	CELL_LC401_AP_TH_D02                            :=      47382       ,
	CELL_LC401_AP_TH_D03                            :=      47383       ,
	CELL_LC401_AP_TH_D04                            :=      47384       ,
	CELL_LC501_TESTER                               :=      47400       ,
	CELL_LC501_TESTER_SOCKET_A01                    :=      47401       ,
	CELL_LC501_TESTER_SOCKET_A02                    :=      47402       ,
	CELL_LC501_TESTER_SOCKET_A03                    :=      47403       ,
	CELL_LC501_TESTER_SOCKET_A04                    :=      47404       ,
	CELL_LC501_TESTER_SOCKET_B01                    :=      47411       ,
	CELL_LC501_TESTER_SOCKET_B02                    :=      47412       ,
	CELL_LC501_TESTER_SOCKET_B03                    :=      47413       ,
	CELL_LC501_TESTER_SOCKET_B04                    :=      47414       ,
	CELL_LC501_TESTER_SOCKET_C01                    :=      47421       ,
	CELL_LC501_TESTER_SOCKET_C02                    :=      47422       ,
	CELL_LC501_TESTER_SOCKET_C03                    :=      47423       ,
	CELL_LC501_TESTER_SOCKET_C04                    :=      47424       ,
	CELL_LC501_TESTER_SOCKET_D01                    :=      47431       ,
	CELL_LC501_TESTER_SOCKET_D02                    :=      47432       ,
	CELL_LC501_TESTER_SOCKET_D03                    :=      47433       ,
	CELL_LC501_TESTER_SOCKET_D04                    :=      47434       ,
	CELL_LC501_AP                                   :=      47450       ,
	CELL_LC501_AP_TH_A01                            :=      47451       ,
	CELL_LC501_AP_TH_A02                            :=      47452       ,
	CELL_LC501_AP_TH_A03                            :=      47453       ,
	CELL_LC501_AP_TH_A04                            :=      47454       ,
	CELL_LC501_AP_TH_B01                            :=      47461       ,
	CELL_LC501_AP_TH_B02                            :=      47462       ,
	CELL_LC501_AP_TH_B03                            :=      47463       ,
	CELL_LC501_AP_TH_B04                            :=      47464       ,
	CELL_LC501_AP_TH_C01                            :=      47471       ,
	CELL_LC501_AP_TH_C02                            :=      47472       ,
	CELL_LC501_AP_TH_C03                            :=      47473       ,
	CELL_LC501_AP_TH_C04                            :=      47474       ,
	CELL_LC501_AP_TH_D01                            :=      47481       ,
	CELL_LC501_AP_TH_D02                            :=      47482       ,
	CELL_LC501_AP_TH_D03                            :=      47483       ,
	CELL_LC501_AP_TH_D04                            :=      47484       ,
	CELL_LC601_TESTER                               :=      47500       ,
	CELL_LC601_TESTER_SOCKET_A01                    :=      47501       ,
	CELL_LC601_TESTER_SOCKET_A02                    :=      47502       ,
	CELL_LC601_TESTER_SOCKET_A03                    :=      47503       ,
	CELL_LC601_TESTER_SOCKET_A04                    :=      47504       ,
	CELL_LC601_TESTER_SOCKET_B01                    :=      47511       ,
	CELL_LC601_TESTER_SOCKET_B02                    :=      47512       ,
	CELL_LC601_TESTER_SOCKET_B03                    :=      47513       ,
	CELL_LC601_TESTER_SOCKET_B04                    :=      47514       ,
	CELL_LC601_TESTER_SOCKET_C01                    :=      47521       ,
	CELL_LC601_TESTER_SOCKET_C02                    :=      47522       ,
	CELL_LC601_TESTER_SOCKET_C03                    :=      47523       ,
	CELL_LC601_TESTER_SOCKET_C04                    :=      47524       ,
	CELL_LC601_TESTER_SOCKET_D01                    :=      47531       ,
	CELL_LC601_TESTER_SOCKET_D02                    :=      47532       ,
	CELL_LC601_TESTER_SOCKET_D03                    :=      47533       ,
	CELL_LC601_TESTER_SOCKET_D04                    :=      47534       ,
	CELL_LC601_AP                                   :=      47550       ,
	CELL_LC601_AP_TH_A01                            :=      47551       ,
	CELL_LC601_AP_TH_A02                            :=      47552       ,
	CELL_LC601_AP_TH_A03                            :=      47553       ,
	CELL_LC601_AP_TH_A04                            :=      47554       ,
	CELL_LC601_AP_TH_B01                            :=      47561       ,
	CELL_LC601_AP_TH_B02                            :=      47562       ,
	CELL_LC601_AP_TH_B03                            :=      47563       ,
	CELL_LC601_AP_TH_B04                            :=      47564       ,
	CELL_LC601_AP_TH_C01                            :=      47571       ,
	CELL_LC601_AP_TH_C02                            :=      47572       ,
	CELL_LC601_AP_TH_C03                            :=      47573       ,
	CELL_LC601_AP_TH_C04                            :=      47574       ,
	CELL_LC601_AP_TH_D01                            :=      47581       ,
	CELL_LC601_AP_TH_D02                            :=      47582       ,
	CELL_LC601_AP_TH_D03                            :=      47583       ,
	CELL_LC601_AP_TH_D04                            :=      47584       ,
	CELL_RA101_TESTER                               :=      50000       ,
	CELL_RA101_TESTER_SOCKET_A01                    :=      50001       ,
	CELL_RA101_TESTER_SOCKET_A02                    :=      50002       ,
	CELL_RA101_TESTER_SOCKET_A03                    :=      50003       ,
	CELL_RA101_TESTER_SOCKET_A04                    :=      50004       ,
	CELL_RA101_TESTER_SOCKET_B01                    :=      50011       ,
	CELL_RA101_TESTER_SOCKET_B02                    :=      50012       ,
	CELL_RA101_TESTER_SOCKET_B03                    :=      50013       ,
	CELL_RA101_TESTER_SOCKET_B04                    :=      50014       ,
	CELL_RA101_TESTER_SOCKET_C01                    :=      50021       ,
	CELL_RA101_TESTER_SOCKET_C02                    :=      50022       ,
	CELL_RA101_TESTER_SOCKET_C03                    :=      50023       ,
	CELL_RA101_TESTER_SOCKET_C04                    :=      50024       ,
	CELL_RA101_TESTER_SOCKET_D01                    :=      50031       ,
	CELL_RA101_TESTER_SOCKET_D02                    :=      50032       ,
	CELL_RA101_TESTER_SOCKET_D03                    :=      50033       ,
	CELL_RA101_TESTER_SOCKET_D04                    :=      50034       ,
	CELL_RA101_AP                                   :=      50050       ,
	CELL_RA101_AP_TH_A01                            :=      50051       ,
	CELL_RA101_AP_TH_A02                            :=      50052       ,
	CELL_RA101_AP_TH_A03                            :=      50053       ,
	CELL_RA101_AP_TH_A04                            :=      50054       ,
	CELL_RA101_AP_TH_B01                            :=      50061       ,
	CELL_RA101_AP_TH_B02                            :=      50062       ,
	CELL_RA101_AP_TH_B03                            :=      50063       ,
	CELL_RA101_AP_TH_B04                            :=      50064       ,
	CELL_RA101_AP_TH_C01                            :=      50071       ,
	CELL_RA101_AP_TH_C02                            :=      50072       ,
	CELL_RA101_AP_TH_C03                            :=      50073       ,
	CELL_RA101_AP_TH_C04                            :=      50074       ,
	CELL_RA101_AP_TH_D01                            :=      50081       ,
	CELL_RA101_AP_TH_D02                            :=      50082       ,
	CELL_RA101_AP_TH_D03                            :=      50083       ,
	CELL_RA101_AP_TH_D04                            :=      50084       ,
	CELL_RA201_TESTER                               :=      50100       ,
	CELL_RA201_TESTER_SOCKET_A01                    :=      50101       ,
	CELL_RA201_TESTER_SOCKET_A02                    :=      50102       ,
	CELL_RA201_TESTER_SOCKET_A03                    :=      50103       ,
	CELL_RA201_TESTER_SOCKET_A04                    :=      50104       ,
	CELL_RA201_TESTER_SOCKET_B01                    :=      50111       ,
	CELL_RA201_TESTER_SOCKET_B02                    :=      50112       ,
	CELL_RA201_TESTER_SOCKET_B03                    :=      50113       ,
	CELL_RA201_TESTER_SOCKET_B04                    :=      50114       ,
	CELL_RA201_TESTER_SOCKET_C01                    :=      50121       ,
	CELL_RA201_TESTER_SOCKET_C02                    :=      50122       ,
	CELL_RA201_TESTER_SOCKET_C03                    :=      50123       ,
	CELL_RA201_TESTER_SOCKET_C04                    :=      50124       ,
	CELL_RA201_TESTER_SOCKET_D01                    :=      50131       ,
	CELL_RA201_TESTER_SOCKET_D02                    :=      50132       ,
	CELL_RA201_TESTER_SOCKET_D03                    :=      50133       ,
	CELL_RA201_TESTER_SOCKET_D04                    :=      50134       ,
	CELL_RA201_AP                                   :=      50150       ,
	CELL_RA201_AP_TH_A01                            :=      50151       ,
	CELL_RA201_AP_TH_A02                            :=      50152       ,
	CELL_RA201_AP_TH_A03                            :=      50153       ,
	CELL_RA201_AP_TH_A04                            :=      50154       ,
	CELL_RA201_AP_TH_B01                            :=      50161       ,
	CELL_RA201_AP_TH_B02                            :=      50162       ,
	CELL_RA201_AP_TH_B03                            :=      50163       ,
	CELL_RA201_AP_TH_B04                            :=      50164       ,
	CELL_RA201_AP_TH_C01                            :=      50171       ,
	CELL_RA201_AP_TH_C02                            :=      50172       ,
	CELL_RA201_AP_TH_C03                            :=      50173       ,
	CELL_RA201_AP_TH_C04                            :=      50174       ,
	CELL_RA201_AP_TH_D01                            :=      50181       ,
	CELL_RA201_AP_TH_D02                            :=      50182       ,
	CELL_RA201_AP_TH_D03                            :=      50183       ,
	CELL_RA201_AP_TH_D04                            :=      50184       ,
	CELL_RA301_TESTER                               :=      50200       ,
	CELL_RA301_TESTER_SOCKET_A01                    :=      50201       ,
	CELL_RA301_TESTER_SOCKET_A02                    :=      50202       ,
	CELL_RA301_TESTER_SOCKET_A03                    :=      50203       ,
	CELL_RA301_TESTER_SOCKET_A04                    :=      50204       ,
	CELL_RA301_TESTER_SOCKET_B01                    :=      50211       ,
	CELL_RA301_TESTER_SOCKET_B02                    :=      50212       ,
	CELL_RA301_TESTER_SOCKET_B03                    :=      50213       ,
	CELL_RA301_TESTER_SOCKET_B04                    :=      50214       ,
	CELL_RA301_TESTER_SOCKET_C01                    :=      50221       ,
	CELL_RA301_TESTER_SOCKET_C02                    :=      50222       ,
	CELL_RA301_TESTER_SOCKET_C03                    :=      50223       ,
	CELL_RA301_TESTER_SOCKET_C04                    :=      50224       ,
	CELL_RA301_TESTER_SOCKET_D01                    :=      50231       ,
	CELL_RA301_TESTER_SOCKET_D02                    :=      50232       ,
	CELL_RA301_TESTER_SOCKET_D03                    :=      50233       ,
	CELL_RA301_TESTER_SOCKET_D04                    :=      50234       ,
	CELL_RA301_AP                                   :=      50250       ,
	CELL_RA301_AP_TH_A01                            :=      50251       ,
	CELL_RA301_AP_TH_A02                            :=      50252       ,
	CELL_RA301_AP_TH_A03                            :=      50253       ,
	CELL_RA301_AP_TH_A04                            :=      50254       ,
	CELL_RA301_AP_TH_B01                            :=      50261       ,
	CELL_RA301_AP_TH_B02                            :=      50262       ,
	CELL_RA301_AP_TH_B03                            :=      50263       ,
	CELL_RA301_AP_TH_B04                            :=      50264       ,
	CELL_RA301_AP_TH_C01                            :=      50271       ,
	CELL_RA301_AP_TH_C02                            :=      50272       ,
	CELL_RA301_AP_TH_C03                            :=      50273       ,
	CELL_RA301_AP_TH_C04                            :=      50274       ,
	CELL_RA301_AP_TH_D01                            :=      50281       ,
	CELL_RA301_AP_TH_D02                            :=      50282       ,
	CELL_RA301_AP_TH_D03                            :=      50283       ,
	CELL_RA301_AP_TH_D04                            :=      50284       ,
	CELL_RA401_TESTER                               :=      50300       ,
	CELL_RA401_TESTER_SOCKET_A01                    :=      50301       ,
	CELL_RA401_TESTER_SOCKET_A02                    :=      50302       ,
	CELL_RA401_TESTER_SOCKET_A03                    :=      50303       ,
	CELL_RA401_TESTER_SOCKET_A04                    :=      50304       ,
	CELL_RA401_TESTER_SOCKET_B01                    :=      50311       ,
	CELL_RA401_TESTER_SOCKET_B02                    :=      50312       ,
	CELL_RA401_TESTER_SOCKET_B03                    :=      50313       ,
	CELL_RA401_TESTER_SOCKET_B04                    :=      50314       ,
	CELL_RA401_TESTER_SOCKET_C01                    :=      50321       ,
	CELL_RA401_TESTER_SOCKET_C02                    :=      50322       ,
	CELL_RA401_TESTER_SOCKET_C03                    :=      50323       ,
	CELL_RA401_TESTER_SOCKET_C04                    :=      50324       ,
	CELL_RA401_TESTER_SOCKET_D01                    :=      50331       ,
	CELL_RA401_TESTER_SOCKET_D02                    :=      50332       ,
	CELL_RA401_TESTER_SOCKET_D03                    :=      50333       ,
	CELL_RA401_TESTER_SOCKET_D04                    :=      50334       ,
	CELL_RA401_AP                                   :=      50350       ,
	CELL_RA401_AP_TH_A01                            :=      50351       ,
	CELL_RA401_AP_TH_A02                            :=      50352       ,
	CELL_RA401_AP_TH_A03                            :=      50353       ,
	CELL_RA401_AP_TH_A04                            :=      50354       ,
	CELL_RA401_AP_TH_B01                            :=      50361       ,
	CELL_RA401_AP_TH_B02                            :=      50362       ,
	CELL_RA401_AP_TH_B03                            :=      50363       ,
	CELL_RA401_AP_TH_B04                            :=      50364       ,
	CELL_RA401_AP_TH_C01                            :=      50371       ,
	CELL_RA401_AP_TH_C02                            :=      50372       ,
	CELL_RA401_AP_TH_C03                            :=      50373       ,
	CELL_RA401_AP_TH_C04                            :=      50374       ,
	CELL_RA401_AP_TH_D01                            :=      50381       ,
	CELL_RA401_AP_TH_D02                            :=      50382       ,
	CELL_RA401_AP_TH_D03                            :=      50383       ,
	CELL_RA401_AP_TH_D04                            :=      50384       ,
	CELL_RA501_TESTER                               :=      50400       ,
	CELL_RA501_TESTER_SOCKET_A01                    :=      50401       ,
	CELL_RA501_TESTER_SOCKET_A02                    :=      50402       ,
	CELL_RA501_TESTER_SOCKET_A03                    :=      50403       ,
	CELL_RA501_TESTER_SOCKET_A04                    :=      50404       ,
	CELL_RA501_TESTER_SOCKET_B01                    :=      50411       ,
	CELL_RA501_TESTER_SOCKET_B02                    :=      50412       ,
	CELL_RA501_TESTER_SOCKET_B03                    :=      50413       ,
	CELL_RA501_TESTER_SOCKET_B04                    :=      50414       ,
	CELL_RA501_TESTER_SOCKET_C01                    :=      50421       ,
	CELL_RA501_TESTER_SOCKET_C02                    :=      50422       ,
	CELL_RA501_TESTER_SOCKET_C03                    :=      50423       ,
	CELL_RA501_TESTER_SOCKET_C04                    :=      50424       ,
	CELL_RA501_TESTER_SOCKET_D01                    :=      50431       ,
	CELL_RA501_TESTER_SOCKET_D02                    :=      50432       ,
	CELL_RA501_TESTER_SOCKET_D03                    :=      50433       ,
	CELL_RA501_TESTER_SOCKET_D04                    :=      50434       ,
	CELL_RA501_AP                                   :=      50450       ,
	CELL_RA501_AP_TH_A01                            :=      50451       ,
	CELL_RA501_AP_TH_A02                            :=      50452       ,
	CELL_RA501_AP_TH_A03                            :=      50453       ,
	CELL_RA501_AP_TH_A04                            :=      50454       ,
	CELL_RA501_AP_TH_B01                            :=      50461       ,
	CELL_RA501_AP_TH_B02                            :=      50462       ,
	CELL_RA501_AP_TH_B03                            :=      50463       ,
	CELL_RA501_AP_TH_B04                            :=      50464       ,
	CELL_RA501_AP_TH_C01                            :=      50471       ,
	CELL_RA501_AP_TH_C02                            :=      50472       ,
	CELL_RA501_AP_TH_C03                            :=      50473       ,
	CELL_RA501_AP_TH_C04                            :=      50474       ,
	CELL_RA501_AP_TH_D01                            :=      50481       ,
	CELL_RA501_AP_TH_D02                            :=      50482       ,
	CELL_RA501_AP_TH_D03                            :=      50483       ,
	CELL_RA501_AP_TH_D04                            :=      50484       ,
	CELL_RA601_TESTER                               :=      50500       ,
	CELL_RA601_TESTER_SOCKET_A01                    :=      50501       ,
	CELL_RA601_TESTER_SOCKET_A02                    :=      50502       ,
	CELL_RA601_TESTER_SOCKET_A03                    :=      50503       ,
	CELL_RA601_TESTER_SOCKET_A04                    :=      50504       ,
	CELL_RA601_TESTER_SOCKET_B01                    :=      50511       ,
	CELL_RA601_TESTER_SOCKET_B02                    :=      50512       ,
	CELL_RA601_TESTER_SOCKET_B03                    :=      50513       ,
	CELL_RA601_TESTER_SOCKET_B04                    :=      50514       ,
	CELL_RA601_TESTER_SOCKET_C01                    :=      50521       ,
	CELL_RA601_TESTER_SOCKET_C02                    :=      50522       ,
	CELL_RA601_TESTER_SOCKET_C03                    :=      50523       ,
	CELL_RA601_TESTER_SOCKET_C04                    :=      50524       ,
	CELL_RA601_TESTER_SOCKET_D01                    :=      50531       ,
	CELL_RA601_TESTER_SOCKET_D02                    :=      50532       ,
	CELL_RA601_TESTER_SOCKET_D03                    :=      50533       ,
	CELL_RA601_TESTER_SOCKET_D04                    :=      50534       ,
	CELL_RA601_AP                                   :=      50550       ,
	CELL_RA601_AP_TH_A01                            :=      50551       ,
	CELL_RA601_AP_TH_A02                            :=      50552       ,
	CELL_RA601_AP_TH_A03                            :=      50553       ,
	CELL_RA601_AP_TH_A04                            :=      50554       ,
	CELL_RA601_AP_TH_B01                            :=      50561       ,
	CELL_RA601_AP_TH_B02                            :=      50562       ,
	CELL_RA601_AP_TH_B03                            :=      50563       ,
	CELL_RA601_AP_TH_B04                            :=      50564       ,
	CELL_RA601_AP_TH_C01                            :=      50571       ,
	CELL_RA601_AP_TH_C02                            :=      50572       ,
	CELL_RA601_AP_TH_C03                            :=      50573       ,
	CELL_RA601_AP_TH_C04                            :=      50574       ,
	CELL_RA601_AP_TH_D01                            :=      50581       ,
	CELL_RA601_AP_TH_D02                            :=      50582       ,
	CELL_RA601_AP_TH_D03                            :=      50583       ,
	CELL_RA601_AP_TH_D04                            :=      50584       ,
	CELL_RB101_TESTER                               :=      51000       ,
	CELL_RB101_TESTER_SOCKET_A01                    :=      51001       ,
	CELL_RB101_TESTER_SOCKET_A02                    :=      51002       ,
	CELL_RB101_TESTER_SOCKET_A03                    :=      51003       ,
	CELL_RB101_TESTER_SOCKET_A04                    :=      51004       ,
	CELL_RB101_TESTER_SOCKET_B01                    :=      51011       ,
	CELL_RB101_TESTER_SOCKET_B02                    :=      51012       ,
	CELL_RB101_TESTER_SOCKET_B03                    :=      51013       ,
	CELL_RB101_TESTER_SOCKET_B04                    :=      51014       ,
	CELL_RB101_TESTER_SOCKET_C01                    :=      51021       ,
	CELL_RB101_TESTER_SOCKET_C02                    :=      51022       ,
	CELL_RB101_TESTER_SOCKET_C03                    :=      51023       ,
	CELL_RB101_TESTER_SOCKET_C04                    :=      51024       ,
	CELL_RB101_TESTER_SOCKET_D01                    :=      51031       ,
	CELL_RB101_TESTER_SOCKET_D02                    :=      51032       ,
	CELL_RB101_TESTER_SOCKET_D03                    :=      51033       ,
	CELL_RB101_TESTER_SOCKET_D04                    :=      51034       ,
	CELL_RB101_AP                                   :=      51050       ,
	CELL_RB101_AP_TH_A01                            :=      51051       ,
	CELL_RB101_AP_TH_A02                            :=      51052       ,
	CELL_RB101_AP_TH_A03                            :=      51053       ,
	CELL_RB101_AP_TH_A04                            :=      51054       ,
	CELL_RB101_AP_TH_B01                            :=      51061       ,
	CELL_RB101_AP_TH_B02                            :=      51062       ,
	CELL_RB101_AP_TH_B03                            :=      51063       ,
	CELL_RB101_AP_TH_B04                            :=      51064       ,
	CELL_RB101_AP_TH_C01                            :=      51071       ,
	CELL_RB101_AP_TH_C02                            :=      51072       ,
	CELL_RB101_AP_TH_C03                            :=      51073       ,
	CELL_RB101_AP_TH_C04                            :=      51074       ,
	CELL_RB101_AP_TH_D01                            :=      51081       ,
	CELL_RB101_AP_TH_D02                            :=      51082       ,
	CELL_RB101_AP_TH_D03                            :=      51083       ,
	CELL_RB101_AP_TH_D04                            :=      51084       ,
	CELL_RB201_TESTER                               :=      51100       ,
	CELL_RB201_TESTER_SOCKET_A01                    :=      51101       ,
	CELL_RB201_TESTER_SOCKET_A02                    :=      51102       ,
	CELL_RB201_TESTER_SOCKET_A03                    :=      51103       ,
	CELL_RB201_TESTER_SOCKET_A04                    :=      51104       ,
	CELL_RB201_TESTER_SOCKET_B01                    :=      51111       ,
	CELL_RB201_TESTER_SOCKET_B02                    :=      51112       ,
	CELL_RB201_TESTER_SOCKET_B03                    :=      51113       ,
	CELL_RB201_TESTER_SOCKET_B04                    :=      51114       ,
	CELL_RB201_TESTER_SOCKET_C01                    :=      51121       ,
	CELL_RB201_TESTER_SOCKET_C02                    :=      51122       ,
	CELL_RB201_TESTER_SOCKET_C03                    :=      51123       ,
	CELL_RB201_TESTER_SOCKET_C04                    :=      51124       ,
	CELL_RB201_TESTER_SOCKET_D01                    :=      51131       ,
	CELL_RB201_TESTER_SOCKET_D02                    :=      51132       ,
	CELL_RB201_TESTER_SOCKET_D03                    :=      51133       ,
	CELL_RB201_TESTER_SOCKET_D04                    :=      51134       ,
	CELL_RB201_AP                                   :=      51150       ,
	CELL_RB201_AP_TH_A01                            :=      51151       ,
	CELL_RB201_AP_TH_A02                            :=      51152       ,
	CELL_RB201_AP_TH_A03                            :=      51153       ,
	CELL_RB201_AP_TH_A04                            :=      51154       ,
	CELL_RB201_AP_TH_B01                            :=      51161       ,
	CELL_RB201_AP_TH_B02                            :=      51162       ,
	CELL_RB201_AP_TH_B03                            :=      51163       ,
	CELL_RB201_AP_TH_B04                            :=      51164       ,
	CELL_RB201_AP_TH_C01                            :=      51171       ,
	CELL_RB201_AP_TH_C02                            :=      51172       ,
	CELL_RB201_AP_TH_C03                            :=      51173       ,
	CELL_RB201_AP_TH_C04                            :=      51174       ,
	CELL_RB201_AP_TH_D01                            :=      51181       ,
	CELL_RB201_AP_TH_D02                            :=      51182       ,
	CELL_RB201_AP_TH_D03                            :=      51183       ,
	CELL_RB201_AP_TH_D04                            :=      51184       ,
	CELL_RB301_TESTER                               :=      51200       ,
	CELL_RB301_TESTER_SOCKET_A01                    :=      51201       ,
	CELL_RB301_TESTER_SOCKET_A02                    :=      51202       ,
	CELL_RB301_TESTER_SOCKET_A03                    :=      51203       ,
	CELL_RB301_TESTER_SOCKET_A04                    :=      51204       ,
	CELL_RB301_TESTER_SOCKET_B01                    :=      51211       ,
	CELL_RB301_TESTER_SOCKET_B02                    :=      51212       ,
	CELL_RB301_TESTER_SOCKET_B03                    :=      51213       ,
	CELL_RB301_TESTER_SOCKET_B04                    :=      51214       ,
	CELL_RB301_TESTER_SOCKET_C01                    :=      51221       ,
	CELL_RB301_TESTER_SOCKET_C02                    :=      51222       ,
	CELL_RB301_TESTER_SOCKET_C03                    :=      51223       ,
	CELL_RB301_TESTER_SOCKET_C04                    :=      51224       ,
	CELL_RB301_TESTER_SOCKET_D01                    :=      51231       ,
	CELL_RB301_TESTER_SOCKET_D02                    :=      51232       ,
	CELL_RB301_TESTER_SOCKET_D03                    :=      51233       ,
	CELL_RB301_TESTER_SOCKET_D04                    :=      51234       ,
	CELL_RB301_AP                                   :=      51250       ,
	CELL_RB301_AP_TH_A01                            :=      51251       ,
	CELL_RB301_AP_TH_A02                            :=      51252       ,
	CELL_RB301_AP_TH_A03                            :=      51253       ,
	CELL_RB301_AP_TH_A04                            :=      51254       ,
	CELL_RB301_AP_TH_B01                            :=      51261       ,
	CELL_RB301_AP_TH_B02                            :=      51262       ,
	CELL_RB301_AP_TH_B03                            :=      51263       ,
	CELL_RB301_AP_TH_B04                            :=      51264       ,
	CELL_RB301_AP_TH_C01                            :=      51271       ,
	CELL_RB301_AP_TH_C02                            :=      51272       ,
	CELL_RB301_AP_TH_C03                            :=      51273       ,
	CELL_RB301_AP_TH_C04                            :=      51274       ,
	CELL_RB301_AP_TH_D01                            :=      51281       ,
	CELL_RB301_AP_TH_D02                            :=      51282       ,
	CELL_RB301_AP_TH_D03                            :=      51283       ,
	CELL_RB301_AP_TH_D04                            :=      51284       ,
	CELL_RB401_TESTER                               :=      51300       ,
	CELL_RB401_TESTER_SOCKET_A01                    :=      51301       ,
	CELL_RB401_TESTER_SOCKET_A02                    :=      51302       ,
	CELL_RB401_TESTER_SOCKET_A03                    :=      51303       ,
	CELL_RB401_TESTER_SOCKET_A04                    :=      51304       ,
	CELL_RB401_TESTER_SOCKET_B01                    :=      51311       ,
	CELL_RB401_TESTER_SOCKET_B02                    :=      51312       ,
	CELL_RB401_TESTER_SOCKET_B03                    :=      51313       ,
	CELL_RB401_TESTER_SOCKET_B04                    :=      51314       ,
	CELL_RB401_TESTER_SOCKET_C01                    :=      51321       ,
	CELL_RB401_TESTER_SOCKET_C02                    :=      51322       ,
	CELL_RB401_TESTER_SOCKET_C03                    :=      51323       ,
	CELL_RB401_TESTER_SOCKET_C04                    :=      51324       ,
	CELL_RB401_TESTER_SOCKET_D01                    :=      51331       ,
	CELL_RB401_TESTER_SOCKET_D02                    :=      51332       ,
	CELL_RB401_TESTER_SOCKET_D03                    :=      51333       ,
	CELL_RB401_TESTER_SOCKET_D04                    :=      51334       ,
	CELL_RB401_AP                                   :=      51350       ,
	CELL_RB401_AP_TH_A01                            :=      51351       ,
	CELL_RB401_AP_TH_A02                            :=      51352       ,
	CELL_RB401_AP_TH_A03                            :=      51353       ,
	CELL_RB401_AP_TH_A04                            :=      51354       ,
	CELL_RB401_AP_TH_B01                            :=      51361       ,
	CELL_RB401_AP_TH_B02                            :=      51362       ,
	CELL_RB401_AP_TH_B03                            :=      51363       ,
	CELL_RB401_AP_TH_B04                            :=      51364       ,
	CELL_RB401_AP_TH_C01                            :=      51371       ,
	CELL_RB401_AP_TH_C02                            :=      51372       ,
	CELL_RB401_AP_TH_C03                            :=      51373       ,
	CELL_RB401_AP_TH_C04                            :=      51374       ,
	CELL_RB401_AP_TH_D01                            :=      51381       ,
	CELL_RB401_AP_TH_D02                            :=      51382       ,
	CELL_RB401_AP_TH_D03                            :=      51383       ,
	CELL_RB401_AP_TH_D04                            :=      51384       ,
	CELL_RB501_TESTER                               :=      51400       ,
	CELL_RB501_TESTER_SOCKET_A01                    :=      51401       ,
	CELL_RB501_TESTER_SOCKET_A02                    :=      51402       ,
	CELL_RB501_TESTER_SOCKET_A03                    :=      51403       ,
	CELL_RB501_TESTER_SOCKET_A04                    :=      51404       ,
	CELL_RB501_TESTER_SOCKET_B01                    :=      51411       ,
	CELL_RB501_TESTER_SOCKET_B02                    :=      51412       ,
	CELL_RB501_TESTER_SOCKET_B03                    :=      51413       ,
	CELL_RB501_TESTER_SOCKET_B04                    :=      51414       ,
	CELL_RB501_TESTER_SOCKET_C01                    :=      51421       ,
	CELL_RB501_TESTER_SOCKET_C02                    :=      51422       ,
	CELL_RB501_TESTER_SOCKET_C03                    :=      51423       ,
	CELL_RB501_TESTER_SOCKET_C04                    :=      51424       ,
	CELL_RB501_TESTER_SOCKET_D01                    :=      51431       ,
	CELL_RB501_TESTER_SOCKET_D02                    :=      51432       ,
	CELL_RB501_TESTER_SOCKET_D03                    :=      51433       ,
	CELL_RB501_TESTER_SOCKET_D04                    :=      51434       ,
	CELL_RB501_AP                                   :=      51450       ,
	CELL_RB501_AP_TH_A01                            :=      51451       ,
	CELL_RB501_AP_TH_A02                            :=      51452       ,
	CELL_RB501_AP_TH_A03                            :=      51453       ,
	CELL_RB501_AP_TH_A04                            :=      51454       ,
	CELL_RB501_AP_TH_B01                            :=      51461       ,
	CELL_RB501_AP_TH_B02                            :=      51462       ,
	CELL_RB501_AP_TH_B03                            :=      51463       ,
	CELL_RB501_AP_TH_B04                            :=      51464       ,
	CELL_RB501_AP_TH_C01                            :=      51471       ,
	CELL_RB501_AP_TH_C02                            :=      51472       ,
	CELL_RB501_AP_TH_C03                            :=      51473       ,
	CELL_RB501_AP_TH_C04                            :=      51474       ,
	CELL_RB501_AP_TH_D01                            :=      51481       ,
	CELL_RB501_AP_TH_D02                            :=      51482       ,
	CELL_RB501_AP_TH_D03                            :=      51483       ,
	CELL_RB501_AP_TH_D04                            :=      51484       ,
	CELL_RB601_TESTER                               :=      51500       ,
	CELL_RB601_TESTER_SOCKET_A01                    :=      51501       ,
	CELL_RB601_TESTER_SOCKET_A02                    :=      51502       ,
	CELL_RB601_TESTER_SOCKET_A03                    :=      51503       ,
	CELL_RB601_TESTER_SOCKET_A04                    :=      51504       ,
	CELL_RB601_TESTER_SOCKET_B01                    :=      51511       ,
	CELL_RB601_TESTER_SOCKET_B02                    :=      51512       ,
	CELL_RB601_TESTER_SOCKET_B03                    :=      51513       ,
	CELL_RB601_TESTER_SOCKET_B04                    :=      51514       ,
	CELL_RB601_TESTER_SOCKET_C01                    :=      51521       ,
	CELL_RB601_TESTER_SOCKET_C02                    :=      51522       ,
	CELL_RB601_TESTER_SOCKET_C03                    :=      51523       ,
	CELL_RB601_TESTER_SOCKET_C04                    :=      51524       ,
	CELL_RB601_TESTER_SOCKET_D01                    :=      51531       ,
	CELL_RB601_TESTER_SOCKET_D02                    :=      51532       ,
	CELL_RB601_TESTER_SOCKET_D03                    :=      51533       ,
	CELL_RB601_TESTER_SOCKET_D04                    :=      51534       ,
	CELL_RB601_AP                                   :=      51550       ,
	CELL_RB601_AP_TH_A01                            :=      51551       ,
	CELL_RB601_AP_TH_A02                            :=      51552       ,
	CELL_RB601_AP_TH_A03                            :=      51553       ,
	CELL_RB601_AP_TH_A04                            :=      51554       ,
	CELL_RB601_AP_TH_B01                            :=      51561       ,
	CELL_RB601_AP_TH_B02                            :=      51562       ,
	CELL_RB601_AP_TH_B03                            :=      51563       ,
	CELL_RB601_AP_TH_B04                            :=      51564       ,
	CELL_RB601_AP_TH_C01                            :=      51571       ,
	CELL_RB601_AP_TH_C02                            :=      51572       ,
	CELL_RB601_AP_TH_C03                            :=      51573       ,
	CELL_RB601_AP_TH_C04                            :=      51574       ,
	CELL_RB601_AP_TH_D01                            :=      51581       ,
	CELL_RB601_AP_TH_D02                            :=      51582       ,
	CELL_RB601_AP_TH_D03                            :=      51583       ,
	CELL_RB601_AP_TH_D04                            :=      51584       ,
	CELL_RC101_TESTER                               :=      52000       ,
	CELL_RC101_TESTER_SOCKET_A01                    :=      52001       ,
	CELL_RC101_TESTER_SOCKET_A02                    :=      52002       ,
	CELL_RC101_TESTER_SOCKET_A03                    :=      52003       ,
	CELL_RC101_TESTER_SOCKET_A04                    :=      52004       ,
	CELL_RC101_TESTER_SOCKET_B01                    :=      52011       ,
	CELL_RC101_TESTER_SOCKET_B02                    :=      52012       ,
	CELL_RC101_TESTER_SOCKET_B03                    :=      52013       ,
	CELL_RC101_TESTER_SOCKET_B04                    :=      52014       ,
	CELL_RC101_TESTER_SOCKET_C01                    :=      52021       ,
	CELL_RC101_TESTER_SOCKET_C02                    :=      52022       ,
	CELL_RC101_TESTER_SOCKET_C03                    :=      52023       ,
	CELL_RC101_TESTER_SOCKET_C04                    :=      52024       ,
	CELL_RC101_TESTER_SOCKET_D01                    :=      52031       ,
	CELL_RC101_TESTER_SOCKET_D02                    :=      52032       ,
	CELL_RC101_TESTER_SOCKET_D03                    :=      52033       ,
	CELL_RC101_TESTER_SOCKET_D04                    :=      52034       ,
	CELL_RC101_AP                                   :=      52050       ,
	CELL_RC101_AP_TH_A01                            :=      52051       ,
	CELL_RC101_AP_TH_A02                            :=      52052       ,
	CELL_RC101_AP_TH_A03                            :=      52053       ,
	CELL_RC101_AP_TH_A04                            :=      52054       ,
	CELL_RC101_AP_TH_B01                            :=      52061       ,
	CELL_RC101_AP_TH_B02                            :=      52062       ,
	CELL_RC101_AP_TH_B03                            :=      52063       ,
	CELL_RC101_AP_TH_B04                            :=      52064       ,
	CELL_RC101_AP_TH_C01                            :=      52071       ,
	CELL_RC101_AP_TH_C02                            :=      52072       ,
	CELL_RC101_AP_TH_C03                            :=      52073       ,
	CELL_RC101_AP_TH_C04                            :=      52074       ,
	CELL_RC101_AP_TH_D01                            :=      52081       ,
	CELL_RC101_AP_TH_D02                            :=      52082       ,
	CELL_RC101_AP_TH_D03                            :=      52083       ,
	CELL_RC101_AP_TH_D04                            :=      52084       ,
	CELL_RC201_TESTER                               :=      52100       ,
	CELL_RC201_TESTER_SOCKET_A01                    :=      52101       ,
	CELL_RC201_TESTER_SOCKET_A02                    :=      52102       ,
	CELL_RC201_TESTER_SOCKET_A03                    :=      52103       ,
	CELL_RC201_TESTER_SOCKET_A04                    :=      52104       ,
	CELL_RC201_TESTER_SOCKET_B01                    :=      52111       ,
	CELL_RC201_TESTER_SOCKET_B02                    :=      52112       ,
	CELL_RC201_TESTER_SOCKET_B03                    :=      52113       ,
	CELL_RC201_TESTER_SOCKET_B04                    :=      52114       ,
	CELL_RC201_TESTER_SOCKET_C01                    :=      52121       ,
	CELL_RC201_TESTER_SOCKET_C02                    :=      52122       ,
	CELL_RC201_TESTER_SOCKET_C03                    :=      52123       ,
	CELL_RC201_TESTER_SOCKET_C04                    :=      52124       ,
	CELL_RC201_TESTER_SOCKET_D01                    :=      52131       ,
	CELL_RC201_TESTER_SOCKET_D02                    :=      52132       ,
	CELL_RC201_TESTER_SOCKET_D03                    :=      52133       ,
	CELL_RC201_TESTER_SOCKET_D04                    :=      52134       ,
	CELL_RC201_AP                                   :=      52150       ,
	CELL_RC201_AP_TH_A01                            :=      52151       ,
	CELL_RC201_AP_TH_A02                            :=      52152       ,
	CELL_RC201_AP_TH_A03                            :=      52153       ,
	CELL_RC201_AP_TH_A04                            :=      52154       ,
	CELL_RC201_AP_TH_B01                            :=      52161       ,
	CELL_RC201_AP_TH_B02                            :=      52162       ,
	CELL_RC201_AP_TH_B03                            :=      52163       ,
	CELL_RC201_AP_TH_B04                            :=      52164       ,
	CELL_RC201_AP_TH_C01                            :=      52171       ,
	CELL_RC201_AP_TH_C02                            :=      52172       ,
	CELL_RC201_AP_TH_C03                            :=      52173       ,
	CELL_RC201_AP_TH_C04                            :=      52174       ,
	CELL_RC201_AP_TH_D01                            :=      52181       ,
	CELL_RC201_AP_TH_D02                            :=      52182       ,
	CELL_RC201_AP_TH_D03                            :=      52183       ,
	CELL_RC201_AP_TH_D04                            :=      52184       ,
	CELL_RC301_TESTER                               :=      52200       ,
	CELL_RC301_TESTER_SOCKET_A01                    :=      52201       ,
	CELL_RC301_TESTER_SOCKET_A02                    :=      52202       ,
	CELL_RC301_TESTER_SOCKET_A03                    :=      52203       ,
	CELL_RC301_TESTER_SOCKET_A04                    :=      52204       ,
	CELL_RC301_TESTER_SOCKET_B01                    :=      52211       ,
	CELL_RC301_TESTER_SOCKET_B02                    :=      52212       ,
	CELL_RC301_TESTER_SOCKET_B03                    :=      52213       ,
	CELL_RC301_TESTER_SOCKET_B04                    :=      52214       ,
	CELL_RC301_TESTER_SOCKET_C01                    :=      52221       ,
	CELL_RC301_TESTER_SOCKET_C02                    :=      52222       ,
	CELL_RC301_TESTER_SOCKET_C03                    :=      52223       ,
	CELL_RC301_TESTER_SOCKET_C04                    :=      52224       ,
	CELL_RC301_TESTER_SOCKET_D01                    :=      52231       ,
	CELL_RC301_TESTER_SOCKET_D02                    :=      52232       ,
	CELL_RC301_TESTER_SOCKET_D03                    :=      52233       ,
	CELL_RC301_TESTER_SOCKET_D04                    :=      52234       ,
	CELL_RC301_AP                                   :=      52250       ,
	CELL_RC301_AP_TH_A01                            :=      52251       ,
	CELL_RC301_AP_TH_A02                            :=      52252       ,
	CELL_RC301_AP_TH_A03                            :=      52253       ,
	CELL_RC301_AP_TH_A04                            :=      52254       ,
	CELL_RC301_AP_TH_B01                            :=      52261       ,
	CELL_RC301_AP_TH_B02                            :=      52262       ,
	CELL_RC301_AP_TH_B03                            :=      52263       ,
	CELL_RC301_AP_TH_B04                            :=      52264       ,
	CELL_RC301_AP_TH_C01                            :=      52271       ,
	CELL_RC301_AP_TH_C02                            :=      52272       ,
	CELL_RC301_AP_TH_C03                            :=      52273       ,
	CELL_RC301_AP_TH_C04                            :=      52274       ,
	CELL_RC301_AP_TH_D01                            :=      52281       ,
	CELL_RC301_AP_TH_D02                            :=      52282       ,
	CELL_RC301_AP_TH_D03                            :=      52283       ,
	CELL_RC301_AP_TH_D04                            :=      52284       ,
	CELL_RC401_TESTER                               :=      52300       ,
	CELL_RC401_TESTER_SOCKET_A01                    :=      52301       ,
	CELL_RC401_TESTER_SOCKET_A02                    :=      52302       ,
	CELL_RC401_TESTER_SOCKET_A03                    :=      52303       ,
	CELL_RC401_TESTER_SOCKET_A04                    :=      52304       ,
	CELL_RC401_TESTER_SOCKET_B01                    :=      52311       ,
	CELL_RC401_TESTER_SOCKET_B02                    :=      52312       ,
	CELL_RC401_TESTER_SOCKET_B03                    :=      52313       ,
	CELL_RC401_TESTER_SOCKET_B04                    :=      52314       ,
	CELL_RC401_TESTER_SOCKET_C01                    :=      52321       ,
	CELL_RC401_TESTER_SOCKET_C02                    :=      52322       ,
	CELL_RC401_TESTER_SOCKET_C03                    :=      52323       ,
	CELL_RC401_TESTER_SOCKET_C04                    :=      52324       ,
	CELL_RC401_TESTER_SOCKET_D01                    :=      52331       ,
	CELL_RC401_TESTER_SOCKET_D02                    :=      52332       ,
	CELL_RC401_TESTER_SOCKET_D03                    :=      52333       ,
	CELL_RC401_TESTER_SOCKET_D04                    :=      52334       ,
	CELL_RC401_AP                                   :=      52350       ,
	CELL_RC401_AP_TH_A01                            :=      52351       ,
	CELL_RC401_AP_TH_A02                            :=      52352       ,
	CELL_RC401_AP_TH_A03                            :=      52353       ,
	CELL_RC401_AP_TH_A04                            :=      52354       ,
	CELL_RC401_AP_TH_B01                            :=      52361       ,
	CELL_RC401_AP_TH_B02                            :=      52362       ,
	CELL_RC401_AP_TH_B03                            :=      52363       ,
	CELL_RC401_AP_TH_B04                            :=      52364       ,
	CELL_RC401_AP_TH_C01                            :=      52371       ,
	CELL_RC401_AP_TH_C02                            :=      52372       ,
	CELL_RC401_AP_TH_C03                            :=      52373       ,
	CELL_RC401_AP_TH_C04                            :=      52374       ,
	CELL_RC401_AP_TH_D01                            :=      52381       ,
	CELL_RC401_AP_TH_D02                            :=      52382       ,
	CELL_RC401_AP_TH_D03                            :=      52383       ,
	CELL_RC401_AP_TH_D04                            :=      52384       ,
	CELL_RC501_TESTER                               :=      52400       ,
	CELL_RC501_TESTER_SOCKET_A01                    :=      52401       ,
	CELL_RC501_TESTER_SOCKET_A02                    :=      52402       ,
	CELL_RC501_TESTER_SOCKET_A03                    :=      52403       ,
	CELL_RC501_TESTER_SOCKET_A04                    :=      52404       ,
	CELL_RC501_TESTER_SOCKET_B01                    :=      52411       ,
	CELL_RC501_TESTER_SOCKET_B02                    :=      52412       ,
	CELL_RC501_TESTER_SOCKET_B03                    :=      52413       ,
	CELL_RC501_TESTER_SOCKET_B04                    :=      52414       ,
	CELL_RC501_TESTER_SOCKET_C01                    :=      52421       ,
	CELL_RC501_TESTER_SOCKET_C02                    :=      52422       ,
	CELL_RC501_TESTER_SOCKET_C03                    :=      52423       ,
	CELL_RC501_TESTER_SOCKET_C04                    :=      52424       ,
	CELL_RC501_TESTER_SOCKET_D01                    :=      52431       ,
	CELL_RC501_TESTER_SOCKET_D02                    :=      52432       ,
	CELL_RC501_TESTER_SOCKET_D03                    :=      52433       ,
	CELL_RC501_TESTER_SOCKET_D04                    :=      52434       ,
	CELL_RC501_AP                                   :=      52450       ,
	CELL_RC501_AP_TH_A01                            :=      52451       ,
	CELL_RC501_AP_TH_A02                            :=      52452       ,
	CELL_RC501_AP_TH_A03                            :=      52453       ,
	CELL_RC501_AP_TH_A04                            :=      52454       ,
	CELL_RC501_AP_TH_B01                            :=      52461       ,
	CELL_RC501_AP_TH_B02                            :=      52462       ,
	CELL_RC501_AP_TH_B03                            :=      52463       ,
	CELL_RC501_AP_TH_B04                            :=      52464       ,
	CELL_RC501_AP_TH_C01                            :=      52471       ,
	CELL_RC501_AP_TH_C02                            :=      52472       ,
	CELL_RC501_AP_TH_C03                            :=      52473       ,
	CELL_RC501_AP_TH_C04                            :=      52474       ,
	CELL_RC501_AP_TH_D01                            :=      52481       ,
	CELL_RC501_AP_TH_D02                            :=      52482       ,
	CELL_RC501_AP_TH_D03                            :=      52483       ,
	CELL_RC501_AP_TH_D04                            :=      52484       ,
	CELL_RC601_TESTER                               :=      52500       ,
	CELL_RC601_TESTER_SOCKET_A01                    :=      52501       ,
	CELL_RC601_TESTER_SOCKET_A02                    :=      52502       ,
	CELL_RC601_TESTER_SOCKET_A03                    :=      52503       ,
	CELL_RC601_TESTER_SOCKET_A04                    :=      52504       ,
	CELL_RC601_TESTER_SOCKET_B01                    :=      52511       ,
	CELL_RC601_TESTER_SOCKET_B02                    :=      52512       ,
	CELL_RC601_TESTER_SOCKET_B03                    :=      52513       ,
	CELL_RC601_TESTER_SOCKET_B04                    :=      52514       ,
	CELL_RC601_TESTER_SOCKET_C01                    :=      52521       ,
	CELL_RC601_TESTER_SOCKET_C02                    :=      52522       ,
	CELL_RC601_TESTER_SOCKET_C03                    :=      52523       ,
	CELL_RC601_TESTER_SOCKET_C04                    :=      52524       ,
	CELL_RC601_TESTER_SOCKET_D01                    :=      52531       ,
	CELL_RC601_TESTER_SOCKET_D02                    :=      52532       ,
	CELL_RC601_TESTER_SOCKET_D03                    :=      52533       ,
	CELL_RC601_TESTER_SOCKET_D04                    :=      52534       ,
	CELL_RC601_AP                                   :=      52550       ,
	CELL_RC601_AP_TH_A01                            :=      52551       ,
	CELL_RC601_AP_TH_A02                            :=      52552       ,
	CELL_RC601_AP_TH_A03                            :=      52553       ,
	CELL_RC601_AP_TH_A04                            :=      52554       ,
	CELL_RC601_AP_TH_B01                            :=      52561       ,
	CELL_RC601_AP_TH_B02                            :=      52562       ,
	CELL_RC601_AP_TH_B03                            :=      52563       ,
	CELL_RC601_AP_TH_B04                            :=      52564       ,
	CELL_RC601_AP_TH_C01                            :=      52571       ,
	CELL_RC601_AP_TH_C02                            :=      52572       ,
	CELL_RC601_AP_TH_C03                            :=      52573       ,
	CELL_RC601_AP_TH_C04                            :=      52574       ,
	CELL_RC601_AP_TH_D01                            :=      52581       ,
	CELL_RC601_AP_TH_D02                            :=      52582       ,
	CELL_RC601_AP_TH_D03                            :=      52583       ,
	CELL_RC601_AP_TH_D04                            :=      52584       
                                                    
                                                    
                                                      
*)                                                
                                                     
(*	                                                
    //Old                                                                                             
	NA := 0,                                              
	Standby := 1,                                         
	IOLP := 2,                                            
	PNB := 3,                                             
	TBOT := 4,                                            
	PNB_UPLOOKING_CAMERA := 5,                            
	LP_VISIONSHUTTLE_L := 1500,                           
	LP_VISIONSHUTTLE_R := 1600,                           
	LP_LE := 1900,                                        
	LP_L01 := 1901,                                       
	LP_L02 := 1902,                                       
	LP_RE := 1903,                                        
	LP_R01 := 1904,                                       
	LP_R02 := 1905,                                       
	LP_LE_STACKER_01 := 2000,                             
	LP_LE_STACKER_01_LIFT := 2001,                        
	LP_LE_STACKER_01_STOPPER_01 := 2002,                  
	LP_LE_STACKER_01_STOPPER_02 := 2003,                  
	LP_LE_STACKER_02 := 2050,                             
	LP_LE_STACKER_02_LIFT := 2051,                        
	LP_LE_STACKER_02_STOPPER_01 := 2052,                  
	LP_LE_STACKER_02_STOPPER_02 := 2053,                  
	LP_LE_CONVEYOR := 2200,                               
	LP_LE_CONVEYOR_STACKER_01_PRE := 2250,                
	LP_LE_CONVEYOR_STACKER_01 := 2251,                    
	LP_LE_CONVEYOR_STACKER_01_POST := 2252,               
	LP_LE_CONVEYOR_STACKER_02 := 2300,                    
	LP_L01_STACKER_01 := 3000,                            
	LP_L01_STACKER_01_LIFT := 3001,                       
	LP_L01_STACKER_01_STOPPER_01 := 3002,                 
	LP_L01_STACKER_01_STOPPER_02 := 3003,                 
	LP_L01_STACKER_02 := 3050,                            
	LP_L01_STACKER_02_LIFT := 3051,                       
	LP_L01_STACKER_02_STOPPER_01 := 3052,                 
	LP_L01_STACKER_02_STOPPER_02 := 3053,                 
	LP_L01_STACKER_03 := 3100,                            
	LP_L01_STACKER_03_LIFT := 3101,                       
	LP_L01_STACKER_03_STOPPER_01 := 3102,                 
	LP_L01_STACKER_03_STOPPER_02 := 3103,                 
	LP_L01_CONVEYOR_01 := 3110,                           
	LP_L01_CONVEYOR_02 := 3120,                           
	LP_L01_EPORT := 3130,                                 
	LP_L01_EPORT_STANDBY := 3131,                         
	LP_L01_VISION := 3140,                                
	LP_L01_UPORT := 3151,                                 
	LP_L02_STACKER_01 := 3200,                            
	LP_L02_STACKER_01_LIFT := 3201,                       
	LP_L02_STACKER_01_STOPPER_01 := 3202,                 
	LP_L02_STACKER_01_STOPPER_02 := 3203,                 
	LP_L02_STACKER_02 := 3250,                            
	LP_L02_STACKER_02_LIFT := 3251,                       
	LP_L02_STACKER_02_STOPPER_01 := 3252,                 
	LP_L02_STACKER_02_STOPPER_02 := 3253,                 
	LP_L02_STACKER_03 := 3300,                            
	LP_L02_STACKER_03_LIFT := 3301,                       
	LP_L02_STACKER_03_STOPPER_01 := 3302,                 
	LP_L02_STACKER_03_STOPPER_02 := 3303,                 
	LP_L02_CONVEYOR_01 := 3310,                           
	LP_L02_CONVEYOR_02 := 3320,                           
	LP_L02_EPORT := 3330,                                 
	LP_L02_EPORT_STANDBY := 3331,                         
	LP_L02_VISION := 3340,                                
	LP_L02_UPORT := 3351,                                 
	LP_RE_STACKER_01 := 4000,                             
	LP_RE_STACKER_01_LIFT := 4001,                        
	LP_RE_STACKER_01_STOPPER_01 := 4002,                  
	LP_RE_STACKER_01_STOPPER_02 := 4003,                  
	LP_RE_STACKER_02 := 4050,                             
	LP_RE_STACKER_02_LIFT := 4051,                        
	LP_RE_STACKER_02_STOPPER_01 := 4052,                  
	LP_RE_STACKER_02_STOPPER_02 := 4053,                  
	LP_RE_CONVEYOR := 4200,                               
	LP_RE_CONVEYOR_STACKER_01_PRE := 4250,                
	LP_RE_CONVEYOR_STACKER_01 := 4251,                    
	LP_RE_CONVEYOR_STACKER_01_POST := 4252,               
	LP_RE_CONVEYOR_STACKER_02 := 4300,                    
	LP_R01_STACKER_01 := 5000,                            
	LP_R01_STACKER_01_LIFT := 5001,                       
	LP_R01_STACKER_01_STOPPER_01 := 5002,                 
	LP_R01_STACKER_01_STOPPER_02 := 5003,                 
	LP_R01_STACKER_02 := 5050,                            
	LP_R01_STACKER_02_LIFT := 5051,                       
	LP_R01_STACKER_02_STOPPER_01 := 5052,                 
	LP_R01_STACKER_02_STOPPER_02 := 5053,                 
	LP_R01_STACKER_03 := 5100,                            
	LP_R01_STACKER_03_LIFT := 5101,                       
	LP_R01_STACKER_03_STOPPER_01 := 5102,                 
	LP_R01_STACKER_03_STOPPER_02 := 5103,                 
	LP_R01_CONVEYOR_01 := 5110,                           
	LP_R01_CONVEYOR_02 := 5120,                           
	LP_R01_EPORT := 5130,                                 
	LP_R01_EPORT_STANDBY := 5131,                         
	LP_R01_VISION := 5140,                                
	LP_R01_UPORT := 5151,                           
	LP_R02_STACKER_01 := 5200,                      
	LP_R02_STACKER_01_LIFT := 5201,                 
	LP_R02_STACKER_01_STOPPER_01 := 5202,           
	LP_R02_STACKER_01_STOPPER_02 := 5203,
	LP_R02_STACKER_02 := 5250,
	LP_R02_STACKER_02_LIFT := 5251,
	LP_R02_STACKER_02_STOPPER_01 := 5252,
	LP_R02_STACKER_02_STOPPER_02 := 5253,
	LP_R02_STACKER_03 := 5300,
	LP_R02_STACKER_03_LIFT := 5301,
	LP_R02_STACKER_03_STOPPER_01 := 5302,
	LP_R02_STACKER_03_STOPPER_02 := 5303,
	LP_R02_CONVEYOR_01 := 5310,
	LP_R02_CONVEYOR_02 := 5320,
	LP_R02_EPORT := 5330,
	LP_R02_EPORT_STANDBY := 5331,
	LP_R02_VISION := 5340,
	LP_R02_UPORT := 5351,
	TTS := 10000,
	TTS_01 := 10100,
	TTS_01_SERVICE := 10101,
	TTS_01_PARK := 10102,
	TTS_02 := 10200,
	TTS_02_SERVICE := 10201,
	TTS_03 := 10300,
	TTS_03_SERVICE := 10301,
	TTS_03_PARK := 10302,
	PNB_LANE_01 := 21000,
	PNB_LANE_02 := 21050,
	PNB_LANE_03 := 21150,
	PNB_LANE_04 := 21200,
	PNB_LANE_05 := 21350,
	PNB_LANE_06 := 21400,
	PNB_LANE_07 := 21450,
	PNB_LANE_08 := 21500,
	PNB_GANTRY_01 := 22500,
	PNB_GANTRY_01_PARK := 22501,
	PNB_UPCAM_L := 22502,
	PNB_RFID_L := 22503,
	PNB_GANTRY_01_HEAD_A01 := 22550,
	PNB_GANTRY_01_HEAD_A02 := 22560,
	PNB_GANTRY_01_HEAD_A03 := 22570,
	PNB_GANTRY_01_HEAD_A04 := 22580,
	PNB_GANTRY_02 := 23000,
	PNB_GANTRY_02_PARK := 23001,
	PNB_UPCAM_R := 23002,
	PNB_RFID_R := 23003,
	PNB_GANTRY_02_HEAD_A01 := 23050,
	PNB_GANTRY_02_HEAD_A02 := 23060,
	PNB_GANTRY_02_HEAD_A03 := 23070,
	PNB_GANTRY_02_HEAD_A04 := 23080,
	PRECISOR_UL := 24000,
	PRECISOR_UL_CLEAN := 24001,
	PRECISOR_UL_01 := 24002,
	PRECISOR_UL_02 := 24003,
	PRECISOR_UL_A01_01 := 24011,
	PRECISOR_UL_A01_02 := 24012,
	PRECISOR_UL_A02_01 := 24021,
	PRECISOR_UL_A02_02 := 24022,
	PRECISOR_UL_A03_01 := 24031,
	PRECISOR_UL_A03_02 := 24032,
	PRECISOR_UL_A04_01 := 24041,
	PRECISOR_UL_A04_02 := 24042,
	PRECISOR_UL_B01_01 := 24061,
	PRECISOR_UL_B01_02 := 24062,
	PRECISOR_UL_B02_01 := 24071,
	PRECISOR_UL_B02_02 := 24072,
	PRECISOR_UL_B03_01 := 24081,
	PRECISOR_UL_B03_02 := 24082,
	PRECISOR_UL_B04_01 := 24091,
	PRECISOR_UL_B04_02 := 24092,
	PRECISOR_UL_C01_01 := 24111,
	PRECISOR_UL_C01_02 := 24112,
	PRECISOR_UL_C02_01 := 24121,
	PRECISOR_UL_C02_02 := 24122,
	PRECISOR_UL_C03_01 := 24131,
	PRECISOR_UL_C03_02 := 24132,
	PRECISOR_UL_C04_01 := 24141,
	PRECISOR_UL_C04_02 := 24142,
	PRECISOR_UL_D01_01 := 24161,
	PRECISOR_UL_D01_02 := 24162,
	PRECISOR_UL_D02_01 := 24171,
	PRECISOR_UL_D02_02 := 24172,
	PRECISOR_UL_D03_01 := 24181,
	PRECISOR_UL_D03_02 := 24182,
	PRECISOR_UL_D04_01 := 24191,
	PRECISOR_UL_D04_02 := 24192,
	PRECISOR_UR := 24500,
	PRECISOR_UR_CLEAN := 24501,
	PRECISOR_UR_01 := 24502,
	PRECISOR_UR_02 := 24503,
	PRECISOR_UR_A01_01 := 24511,
	PRECISOR_UR_A01_02 := 24512,
	PRECISOR_UR_A02_01 := 24521,
	PRECISOR_UR_A02_02 := 24522,
	PRECISOR_UR_A03_01 := 24531,
	PRECISOR_UR_A03_02 := 24532,
	PRECISOR_UR_A04_01 := 24541,
	PRECISOR_UR_A04_02 := 24542,
	PRECISOR_UR_B01_01 := 24561,
	PRECISOR_UR_B01_02 := 24562,
	PRECISOR_UR_B02_01 := 24571,
	PRECISOR_UR_B02_02 := 24572,
	PRECISOR_UR_B03_01 := 24581,
	PRECISOR_UR_B03_02 := 24582,
	PRECISOR_UR_B04_01 := 24591,
	PRECISOR_UR_B04_02 := 24592,
	PRECISOR_UR_C01_01 := 24611,
	PRECISOR_UR_C01_02 := 24612,
	PRECISOR_UR_C02_01 := 24621,
	PRECISOR_UR_C02_02 := 24622,
	PRECISOR_UR_C03_01 := 24631,
	PRECISOR_UR_C03_02 := 24632,
	PRECISOR_UR_C04_01 := 24641,
	PRECISOR_UR_C04_02 := 24642,
	PRECISOR_UR_D01_01 := 24661,
	PRECISOR_UR_D01_02 := 24662,
	PRECISOR_UR_D02_01 := 24671,
	PRECISOR_UR_D02_02 := 24672,
	PRECISOR_UR_D03_01 := 24681,
	PRECISOR_UR_D03_02 := 24682,
	PRECISOR_UR_D04_01 := 24691,
	PRECISOR_UR_D04_02 := 24692,
	PRECISOR_DL := 25000,
	PRECISOR_DL_CLEAN := 25001,
	PRECISOR_DL_01 := 25002,
	PRECISOR_DL_02 := 25003,
	PRECISOR_DL_A01_01 := 25011,
	PRECISOR_DL_A01_02 := 25012,
	PRECISOR_DL_A02_01 := 25021,
	PRECISOR_DL_A02_02 := 25022,
	PRECISOR_DL_A03_01 := 25031,
	PRECISOR_DL_A03_02 := 25032,
	PRECISOR_DL_A04_01 := 25041,
	PRECISOR_DL_A04_02 := 25042,
	PRECISOR_DL_B01_01 := 25061,
	PRECISOR_DL_B01_02 := 25062,
	PRECISOR_DL_B02_01 := 25071,
	PRECISOR_DL_B02_02 := 25072,
	PRECISOR_DL_B03_01 := 25081,
	PRECISOR_DL_B03_02 := 25082,
	PRECISOR_DL_B04_01 := 25091,
	PRECISOR_DL_B04_02 := 25092,
	PRECISOR_DL_C01_01 := 25111,
	PRECISOR_DL_C01_02 := 25112,
	PRECISOR_DL_C02_01 := 25121,
	PRECISOR_DL_C02_02 := 25122,
	PRECISOR_DL_C03_01 := 25131,
	PRECISOR_DL_C03_02 := 25132,
	PRECISOR_DL_C04_01 := 25141,
	PRECISOR_DL_C04_02 := 25142,
	PRECISOR_DL_D01_01 := 25161,
	PRECISOR_DL_D01_02 := 25162,
	PRECISOR_DL_D02_01 := 25171,
	PRECISOR_DL_D02_02 := 25172,
	PRECISOR_DL_D03_01 := 25181,
	PRECISOR_DL_D03_02 := 25182,
	PRECISOR_DL_D04_01 := 25191,
	PRECISOR_DL_D04_02 := 25192,
	PRECISOR_DR := 25500,
	PRECISOR_DR_CLEAN := 25501,
	PRECISOR_DR_01 := 25502,
	PRECISOR_DR_02 := 25503,
	PRECISOR_DR_A01_01 := 25511,
	PRECISOR_DR_A01_02 := 25512,
	PRECISOR_DR_A02_01 := 25521,
	PRECISOR_DR_A02_02 := 25522,
	PRECISOR_DR_A03_01 := 25531,
	PRECISOR_DR_A03_02 := 25532,
	PRECISOR_DR_A04_01 := 25541,
	PRECISOR_DR_A04_02 := 25542,
	PRECISOR_DR_B01_01 := 25561,
	PRECISOR_DR_B01_02 := 25562,
	PRECISOR_DR_B02_01 := 25571,
	PRECISOR_DR_B02_02 := 25572,
	PRECISOR_DR_B03_01 := 25581,
	PRECISOR_DR_B03_02 := 25582,
	PRECISOR_DR_B04_01 := 25591,
	PRECISOR_DR_B04_02 := 25592,
	PRECISOR_DR_C01_01 := 25611,
	PRECISOR_DR_C01_02 := 25612,
	PRECISOR_DR_C02_01 := 25621,
	PRECISOR_DR_C02_02 := 25622,
	PRECISOR_DR_C03_01 := 25631,
	PRECISOR_DR_C03_02 := 25632,
	PRECISOR_DR_C04_01 := 25641,
	PRECISOR_DR_C04_02 := 25642,
	PRECISOR_DR_D01_01 := 25661,
	PRECISOR_DR_D01_02 := 25662,
	PRECISOR_DR_D02_01 := 25671,
	PRECISOR_DR_D02_02 := 25672,
	PRECISOR_DR_D03_01 := 25681,
	PRECISOR_DR_D03_02 := 25682,
	PRECISOR_DR_D04_01 := 25691,
	PRECISOR_DR_D04_02 := 25692,
	TBOT_L := 30000,
	TBOT_L_RFID := 30001,
	TBOT_L_SERVICE := 30002,
	TBOT_L_HEAD_A01 := 30020,
	TBOT_L_HEAD_A02 := 30040,
	TBOT_L_HEAD_A03 := 30060,
	TBOT_L_HEAD_A04 := 30080,
	TBOT_L_HEAD_B01 := 30100,
	TBOT_L_HEAD_B02 := 30120,
	TBOT_L_HEAD_B03 := 30140,
	TBOT_L_HEAD_B04 := 30160,
	TBOT_L_HEAD_C01 := 30180,
	TBOT_L_HEAD_C02 := 30200,
	TBOT_L_HEAD_C03 := 30220,
	TBOT_L_HEAD_C04 := 30240,
	TBOT_L_HEAD_D01 := 30260,
	TBOT_L_HEAD_D02 := 30280,
	TBOT_L_HEAD_D03 := 30300,
	TBOT_L_HEAD_D04 := 30320,
	TBOT_R := 30500,
	TBOT_R_RFID := 30501,
	TBOT_R_SERVICE := 30502,
	TBOT_R_HEAD_A01 := 30520,
	TBOT_R_HEAD_A02 := 30540,
	TBOT_R_HEAD_A03 := 30560,
	TBOT_R_HEAD_A04 := 30580,
	TBOT_R_HEAD_B01 := 30600,
	TBOT_R_HEAD_B02 := 30620,
	TBOT_R_HEAD_B03 := 30640,
	TBOT_R_HEAD_B04 := 30660,
	TBOT_R_HEAD_C01 := 30680,
	TBOT_R_HEAD_C02 := 30700,
	TBOT_R_HEAD_C03 := 30720,
	TBOT_R_HEAD_C04 := 30740,
	TBOT_R_HEAD_D01 := 30760,
	TBOT_R_HEAD_D02 := 30780,
	TBOT_R_HEAD_D03 := 30800,
	TBOT_R_HEAD_D04 := 30820,
	COLUMN_LA := 35000,
	COLUMN_LB := 35100,
	COLUMN_LC := 35200,
	COLUMN_RA := 35300,
	COLUMN_RB := 35400,
	COLUMN_RC := 35500,
	TESTER_LA01 := 45000,
	TESTER_LA01_SOCKET_A01 := 45001,
	TESTER_LA01_SOCKET_A02 := 45002,
	TESTER_LA01_SOCKET_A03 := 45003,
	TESTER_LA01_SOCKET_A04 := 45004,
	TESTER_LA01_SOCKET_B01 := 45011,
	TESTER_LA01_SOCKET_B02 := 45012,
	TESTER_LA01_SOCKET_B03 := 45013,
	TESTER_LA01_SOCKET_B04 := 45014,
	TESTER_LA01_SOCKET_C01 := 45021,
	TESTER_LA01_SOCKET_C02 := 45022,
	TESTER_LA01_SOCKET_C03 := 45023,
	TESTER_LA01_SOCKET_C04 := 45024,
	TESTER_LA01_SOCKET_D01 := 45031,
	TESTER_LA01_SOCKET_D02 := 45032,
	TESTER_LA01_SOCKET_D03 := 45033,
	TESTER_LA01_SOCKET_D04 := 45034,
	TESTER_LA01_TH_A01 := 45051,
	TESTER_LA01_TH_A02 := 45052,
	TESTER_LA01_TH_A03 := 45053,
	TESTER_LA01_TH_A04 := 45054,
	TESTER_LA01_TH_B01 := 45061,
	TESTER_LA01_TH_B02 := 45062,
	TESTER_LA01_TH_B03 := 45063,
	TESTER_LA01_TH_B04 := 45064,
	TESTER_LA01_TH_C01 := 45071,
	TESTER_LA01_TH_C02 := 45072,
	TESTER_LA01_TH_C03 := 45073,
	TESTER_LA01_TH_C04 := 45074,
	TESTER_LA01_TH_D01 := 45081,
	TESTER_LA01_TH_D02 := 45082,
	TESTER_LA01_TH_D03 := 45083,
	TESTER_LA01_TH_D04 := 45084,
	TESTER_LA02 := 45100,
	TESTER_LA02_SOCKET_A01 := 45101,
	TESTER_LA02_SOCKET_A02 := 45102,
	TESTER_LA02_SOCKET_A03 := 45103,
	TESTER_LA02_SOCKET_A04 := 45104,
	TESTER_LA02_SOCKET_B01 := 45111,
	TESTER_LA02_SOCKET_B02 := 45112,
	TESTER_LA02_SOCKET_B03 := 45113,
	TESTER_LA02_SOCKET_B04 := 45114,
	TESTER_LA02_SOCKET_C01 := 45121,
	TESTER_LA02_SOCKET_C02 := 45122,
	TESTER_LA02_SOCKET_C03 := 45123,
	TESTER_LA02_SOCKET_C04 := 45124,
	TESTER_LA02_SOCKET_D01 := 45131,
	TESTER_LA02_SOCKET_D02 := 45132,
	TESTER_LA02_SOCKET_D03 := 45133,
	TESTER_LA02_SOCKET_D04 := 45134,
	TESTER_LA02_TH_A01 := 45151,
	TESTER_LA02_TH_A02 := 45152,
	TESTER_LA02_TH_A03 := 45153,
	TESTER_LA02_TH_A04 := 45154,
	TESTER_LA02_TH_B01 := 45161,
	TESTER_LA02_TH_B02 := 45162,
	TESTER_LA02_TH_B03 := 45163,
	TESTER_LA02_TH_B04 := 45164,
	TESTER_LA02_TH_C01 := 45171,
	TESTER_LA02_TH_C02 := 45172,
	TESTER_LA02_TH_C03 := 45173,
	TESTER_LA02_TH_C04 := 45174,
	TESTER_LA02_TH_D01 := 45181,
	TESTER_LA02_TH_D02 := 45182,
	TESTER_LA02_TH_D03 := 45183,
	TESTER_LA02_TH_D04 := 45184,
	TESTER_LA03 := 45200,
	TESTER_LA03_SOCKET_A01 := 45201,
	TESTER_LA03_SOCKET_A02 := 45202,
	TESTER_LA03_SOCKET_A03 := 45203,
	TESTER_LA03_SOCKET_A04 := 45204,
	TESTER_LA03_SOCKET_B01 := 45211,
	TESTER_LA03_SOCKET_B02 := 45212,
	TESTER_LA03_SOCKET_B03 := 45213,
	TESTER_LA03_SOCKET_B04 := 45214,
	TESTER_LA03_SOCKET_C01 := 45221,
	TESTER_LA03_SOCKET_C02 := 45222,
	TESTER_LA03_SOCKET_C03 := 45223,
	TESTER_LA03_SOCKET_C04 := 45224,
	TESTER_LA03_SOCKET_D01 := 45231,
	TESTER_LA03_SOCKET_D02 := 45232,
	TESTER_LA03_SOCKET_D03 := 45233,
	TESTER_LA03_SOCKET_D04 := 45234,
	TESTER_LA03_TH_A01 := 45251,
	TESTER_LA03_TH_A02 := 45252,
	TESTER_LA03_TH_A03 := 45253,
	TESTER_LA03_TH_A04 := 45254,
	TESTER_LA03_TH_B01 := 45261,
	TESTER_LA03_TH_B02 := 45262,
	TESTER_LA03_TH_B03 := 45263,
	TESTER_LA03_TH_B04 := 45264,
	TESTER_LA03_TH_C01 := 45271,
	TESTER_LA03_TH_C02 := 45272,
	TESTER_LA03_TH_C03 := 45273,
	TESTER_LA03_TH_C04 := 45274,
	TESTER_LA03_TH_D01 := 45281,
	TESTER_LA03_TH_D02 := 45282,
	TESTER_LA03_TH_D03 := 45283,
	TESTER_LA03_TH_D04 := 45284,
	TESTER_LA04 := 45300,
	TESTER_LA04_SOCKET_A01 := 45301,
	TESTER_LA04_SOCKET_A02 := 45302,
	TESTER_LA04_SOCKET_A03 := 45303,
	TESTER_LA04_SOCKET_A04 := 45304,
	TESTER_LA04_SOCKET_B01 := 45311,
	TESTER_LA04_SOCKET_B02 := 45312,
	TESTER_LA04_SOCKET_B03 := 45313,
	TESTER_LA04_SOCKET_B04 := 45314,
	TESTER_LA04_SOCKET_C01 := 45321,
	TESTER_LA04_SOCKET_C02 := 45322,
	TESTER_LA04_SOCKET_C03 := 45323,
	TESTER_LA04_SOCKET_C04 := 45324,
	TESTER_LA04_SOCKET_D01 := 45331,
	TESTER_LA04_SOCKET_D02 := 45332,
	TESTER_LA04_SOCKET_D03 := 45333,
	TESTER_LA04_SOCKET_D04 := 45334,
	TESTER_LA04_TH_A01 := 45351,
	TESTER_LA04_TH_A02 := 45352,
	TESTER_LA04_TH_A03 := 45353,
	TESTER_LA04_TH_A04 := 45354,
	TESTER_LA04_TH_B01 := 45361,
	TESTER_LA04_TH_B02 := 45362,
	TESTER_LA04_TH_B03 := 45363,
	TESTER_LA04_TH_B04 := 45364,
	TESTER_LA04_TH_C01 := 45371,
	TESTER_LA04_TH_C02 := 45372,
	TESTER_LA04_TH_C03 := 45373,
	TESTER_LA04_TH_C04 := 45374,
	TESTER_LA04_TH_D01 := 45381,
	TESTER_LA04_TH_D02 := 45382,
	TESTER_LA04_TH_D03 := 45383,
	TESTER_LA04_TH_D04 := 45384,
	TESTER_LA05 := 45400,
	TESTER_LA05_SOCKET_A01 := 45401,
	TESTER_LA05_SOCKET_A02 := 45402,
	TESTER_LA05_SOCKET_A03 := 45403,
	TESTER_LA05_SOCKET_A04 := 45404,
	TESTER_LA05_SOCKET_B01 := 45411,
	TESTER_LA05_SOCKET_B02 := 45412,
	TESTER_LA05_SOCKET_B03 := 45413,
	TESTER_LA05_SOCKET_B04 := 45414,
	TESTER_LA05_SOCKET_C01 := 45421,
	TESTER_LA05_SOCKET_C02 := 45422,
	TESTER_LA05_SOCKET_C03 := 45423,
	TESTER_LA05_SOCKET_C04 := 45424,
	TESTER_LA05_SOCKET_D01 := 45431,
	TESTER_LA05_SOCKET_D02 := 45432,
	TESTER_LA05_SOCKET_D03 := 45433,
	TESTER_LA05_SOCKET_D04 := 45434,
	TESTER_LA05_TH_A01 := 45451,
	TESTER_LA05_TH_A02 := 45452,
	TESTER_LA05_TH_A03 := 45453,
	TESTER_LA05_TH_A04 := 45454,
	TESTER_LA05_TH_B01 := 45461,
	TESTER_LA05_TH_B02 := 45462,
	TESTER_LA05_TH_B03 := 45463,
	TESTER_LA05_TH_B04 := 45464,
	TESTER_LA05_TH_C01 := 45471,
	TESTER_LA05_TH_C02 := 45472,
	TESTER_LA05_TH_C03 := 45473,
	TESTER_LA05_TH_C04 := 45474,
	TESTER_LA05_TH_D01 := 45481,
	TESTER_LA05_TH_D02 := 45482,
	TESTER_LA05_TH_D03 := 45483,
	TESTER_LA05_TH_D04 := 45484,
	TESTER_LA06 := 45500,
	TESTER_LA06_SOCKET_A01 := 45501,
	TESTER_LA06_SOCKET_A02 := 45502,
	TESTER_LA06_SOCKET_A03 := 45503,
	TESTER_LA06_SOCKET_A04 := 45504,
	TESTER_LA06_SOCKET_B01 := 45511,
	TESTER_LA06_SOCKET_B02 := 45512,
	TESTER_LA06_SOCKET_B03 := 45513,
	TESTER_LA06_SOCKET_B04 := 45514,
	TESTER_LA06_SOCKET_C01 := 45521,
	TESTER_LA06_SOCKET_C02 := 45522,
	TESTER_LA06_SOCKET_C03 := 45523,
	TESTER_LA06_SOCKET_C04 := 45524,
	TESTER_LA06_SOCKET_D01 := 45531,
	TESTER_LA06_SOCKET_D02 := 45532,
	TESTER_LA06_SOCKET_D03 := 45533,
	TESTER_LA06_SOCKET_D04 := 45534,
	TESTER_LA06_TH_A01 := 45551,
	TESTER_LA06_TH_A02 := 45552,
	TESTER_LA06_TH_A03 := 45553,
	TESTER_LA06_TH_A04 := 45554,
	TESTER_LA06_TH_B01 := 45561,
	TESTER_LA06_TH_B02 := 45562,
	TESTER_LA06_TH_B03 := 45563,
	TESTER_LA06_TH_B04 := 45564,
	TESTER_LA06_TH_C01 := 45571,
	TESTER_LA06_TH_C02 := 45572,
	TESTER_LA06_TH_C03 := 45573,
	TESTER_LA06_TH_C04 := 45574,
	TESTER_LA06_TH_D01 := 45581,
	TESTER_LA06_TH_D02 := 45582,
	TESTER_LA06_TH_D03 := 45583,
	TESTER_LA06_TH_D04 := 45584,
	TESTER_LB01 := 46000,
	TESTER_LB01_SOCKET_A01 := 46001,
	TESTER_LB01_SOCKET_A02 := 46002,
	TESTER_LB01_SOCKET_A03 := 46003,
	TESTER_LB01_SOCKET_A04 := 46004,
	TESTER_LB01_SOCKET_B01 := 46011,
	TESTER_LB01_SOCKET_B02 := 46012,
	TESTER_LB01_SOCKET_B03 := 46013,
	TESTER_LB01_SOCKET_B04 := 46014,
	TESTER_LB01_SOCKET_C01 := 46021,
	TESTER_LB01_SOCKET_C02 := 46022,
	TESTER_LB01_SOCKET_C03 := 46023,
	TESTER_LB01_SOCKET_C04 := 46024,
	TESTER_LB01_SOCKET_D01 := 46031,
	TESTER_LB01_SOCKET_D02 := 46032,
	TESTER_LB01_SOCKET_D03 := 46033,
	TESTER_LB01_SOCKET_D04 := 46034,
	TESTER_LB01_TH_A01 := 46051,
	TESTER_LB01_TH_A02 := 46052,
	TESTER_LB01_TH_A03 := 46053,
	TESTER_LB01_TH_A04 := 46054,
	TESTER_LB01_TH_B01 := 46061,
	TESTER_LB01_TH_B02 := 46062,
	TESTER_LB01_TH_B03 := 46063,
	TESTER_LB01_TH_B04 := 46064,
	TESTER_LB01_TH_C01 := 46071,
	TESTER_LB01_TH_C02 := 46072,
	TESTER_LB01_TH_C03 := 46073,
	TESTER_LB01_TH_C04 := 46074,
	TESTER_LB01_TH_D01 := 46081,
	TESTER_LB01_TH_D02 := 46082,
	TESTER_LB01_TH_D03 := 46083,
	TESTER_LB01_TH_D04 := 46084,
	TESTER_LB02 := 46100,
	TESTER_LB02_SOCKET_A01 := 46101,
	TESTER_LB02_SOCKET_A02 := 46102,
	TESTER_LB02_SOCKET_A03 := 46103,
	TESTER_LB02_SOCKET_A04 := 46104,
	TESTER_LB02_SOCKET_B01 := 46111,
	TESTER_LB02_SOCKET_B02 := 46112,
	TESTER_LB02_SOCKET_B03 := 46113,
	TESTER_LB02_SOCKET_B04 := 46114,
	TESTER_LB02_SOCKET_C01 := 46121,
	TESTER_LB02_SOCKET_C02 := 46122,
	TESTER_LB02_SOCKET_C03 := 46123,
	TESTER_LB02_SOCKET_C04 := 46124,
	TESTER_LB02_SOCKET_D01 := 46131,
	TESTER_LB02_SOCKET_D02 := 46132,
	TESTER_LB02_SOCKET_D03 := 46133,
	TESTER_LB02_SOCKET_D04 := 46134,
	TESTER_LB02_TH_A01 := 46151,
	TESTER_LB02_TH_A02 := 46152,
	TESTER_LB02_TH_A03 := 46153,
	TESTER_LB02_TH_A04 := 46154,
	TESTER_LB02_TH_B01 := 46161,
	TESTER_LB02_TH_B02 := 46162,
	TESTER_LB02_TH_B03 := 46163,
	TESTER_LB02_TH_B04 := 46164,
	TESTER_LB02_TH_C01 := 46171,
	TESTER_LB02_TH_C02 := 46172,
	TESTER_LB02_TH_C03 := 46173,
	TESTER_LB02_TH_C04 := 46174,
	TESTER_LB02_TH_D01 := 46181,
	TESTER_LB02_TH_D02 := 46182,
	TESTER_LB02_TH_D03 := 46183,
	TESTER_LB02_TH_D04 := 46184,
	TESTER_LB03 := 46200,
	TESTER_LB03_SOCKET_A01 := 46201,
	TESTER_LB03_SOCKET_A02 := 46202,
	TESTER_LB03_SOCKET_A03 := 46203,
	TESTER_LB03_SOCKET_A04 := 46204,
	TESTER_LB03_SOCKET_B01 := 46211,
	TESTER_LB03_SOCKET_B02 := 46212,
	TESTER_LB03_SOCKET_B03 := 46213,
	TESTER_LB03_SOCKET_B04 := 46214,
	TESTER_LB03_SOCKET_C01 := 46221,
	TESTER_LB03_SOCKET_C02 := 46222,
	TESTER_LB03_SOCKET_C03 := 46223,
	TESTER_LB03_SOCKET_C04 := 46224,
	TESTER_LB03_SOCKET_D01 := 46231,
	TESTER_LB03_SOCKET_D02 := 46232,
	TESTER_LB03_SOCKET_D03 := 46233,
	TESTER_LB03_SOCKET_D04 := 46234,
	TESTER_LB03_TH_A01 := 46251,
	TESTER_LB03_TH_A02 := 46252,
	TESTER_LB03_TH_A03 := 46253,
	TESTER_LB03_TH_A04 := 46254,
	TESTER_LB03_TH_B01 := 46261,
	TESTER_LB03_TH_B02 := 46262,
	TESTER_LB03_TH_B03 := 46263,
	TESTER_LB03_TH_B04 := 46264,
	TESTER_LB03_TH_C01 := 46271,
	TESTER_LB03_TH_C02 := 46272,
	TESTER_LB03_TH_C03 := 46273,
	TESTER_LB03_TH_C04 := 46274,
	TESTER_LB03_TH_D01 := 46281,
	TESTER_LB03_TH_D02 := 46282,
	TESTER_LB03_TH_D03 := 46283,
	TESTER_LB03_TH_D04 := 46284,
	TESTER_LB04 := 46300,
	TESTER_LB04_SOCKET_A01 := 46301,
	TESTER_LB04_SOCKET_A02 := 46302,
	TESTER_LB04_SOCKET_A03 := 46303,
	TESTER_LB04_SOCKET_A04 := 46304,
	TESTER_LB04_SOCKET_B01 := 46311,
	TESTER_LB04_SOCKET_B02 := 46312,
	TESTER_LB04_SOCKET_B03 := 46313,
	TESTER_LB04_SOCKET_B04 := 46314,
	TESTER_LB04_SOCKET_C01 := 46321,
	TESTER_LB04_SOCKET_C02 := 46322,
	TESTER_LB04_SOCKET_C03 := 46323,
	TESTER_LB04_SOCKET_C04 := 46324,
	TESTER_LB04_SOCKET_D01 := 46331,
	TESTER_LB04_SOCKET_D02 := 46332,
	TESTER_LB04_SOCKET_D03 := 46333,
	TESTER_LB04_SOCKET_D04 := 46334,
	TESTER_LB04_TH_A01 := 46351,
	TESTER_LB04_TH_A02 := 46352,
	TESTER_LB04_TH_A03 := 46353,
	TESTER_LB04_TH_A04 := 46354,
	TESTER_LB04_TH_B01 := 46361,
	TESTER_LB04_TH_B02 := 46362,
	TESTER_LB04_TH_B03 := 46363,
	TESTER_LB04_TH_B04 := 46364,
	TESTER_LB04_TH_C01 := 46371,
	TESTER_LB04_TH_C02 := 46372,
	TESTER_LB04_TH_C03 := 46373,
	TESTER_LB04_TH_C04 := 46374,
	TESTER_LB04_TH_D01 := 46381,
	TESTER_LB04_TH_D02 := 46382,
	TESTER_LB04_TH_D03 := 46383,
	TESTER_LB04_TH_D04 := 46384,
	TESTER_LB05 := 46400,
	TESTER_LB05_SOCKET_A01 := 46401,
	TESTER_LB05_SOCKET_A02 := 46402,
	TESTER_LB05_SOCKET_A03 := 46403,
	TESTER_LB05_SOCKET_A04 := 46404,
	TESTER_LB05_SOCKET_B01 := 46411,
	TESTER_LB05_SOCKET_B02 := 46412,
	TESTER_LB05_SOCKET_B03 := 46413,
	TESTER_LB05_SOCKET_B04 := 46414,
	TESTER_LB05_SOCKET_C01 := 46421,
	TESTER_LB05_SOCKET_C02 := 46422,
	TESTER_LB05_SOCKET_C03 := 46423,
	TESTER_LB05_SOCKET_C04 := 46424,
	TESTER_LB05_SOCKET_D01 := 46431,
	TESTER_LB05_SOCKET_D02 := 46432,
	TESTER_LB05_SOCKET_D03 := 46433,
	TESTER_LB05_SOCKET_D04 := 46434,
	TESTER_LB05_TH_A01 := 46451,
	TESTER_LB05_TH_A02 := 46452,
	TESTER_LB05_TH_A03 := 46453,
	TESTER_LB05_TH_A04 := 46454,
	TESTER_LB05_TH_B01 := 46461,
	TESTER_LB05_TH_B02 := 46462,
	TESTER_LB05_TH_B03 := 46463,
	TESTER_LB05_TH_B04 := 46464,
	TESTER_LB05_TH_C01 := 46471,
	TESTER_LB05_TH_C02 := 46472,
	TESTER_LB05_TH_C03 := 46473,
	TESTER_LB05_TH_C04 := 46474,
	TESTER_LB05_TH_D01 := 46481,
	TESTER_LB05_TH_D02 := 46482,
	TESTER_LB05_TH_D03 := 46483,
	TESTER_LB05_TH_D04 := 46484,
	TESTER_LB06 := 46500,
	TESTER_LB06_SOCKET_A01 := 46501,
	TESTER_LB06_SOCKET_A02 := 46502,
	TESTER_LB06_SOCKET_A03 := 46503,
	TESTER_LB06_SOCKET_A04 := 46504,
	TESTER_LB06_SOCKET_B01 := 46511,
	TESTER_LB06_SOCKET_B02 := 46512,
	TESTER_LB06_SOCKET_B03 := 46513,
	TESTER_LB06_SOCKET_B04 := 46514,
	TESTER_LB06_SOCKET_C01 := 46521,
	TESTER_LB06_SOCKET_C02 := 46522,
	TESTER_LB06_SOCKET_C03 := 46523,
	TESTER_LB06_SOCKET_C04 := 46524,
	TESTER_LB06_SOCKET_D01 := 46531,
	TESTER_LB06_SOCKET_D02 := 46532,
	TESTER_LB06_SOCKET_D03 := 46533,
	TESTER_LB06_SOCKET_D04 := 46534,
	TESTER_LB06_TH_A01 := 46551,
	TESTER_LB06_TH_A02 := 46552,
	TESTER_LB06_TH_A03 := 46553,
	TESTER_LB06_TH_A04 := 46554,
	TESTER_LB06_TH_B01 := 46561,
	TESTER_LB06_TH_B02 := 46562,
	TESTER_LB06_TH_B03 := 46563,
	TESTER_LB06_TH_B04 := 46564,
	TESTER_LB06_TH_C01 := 46571,
	TESTER_LB06_TH_C02 := 46572,
	TESTER_LB06_TH_C03 := 46573,
	TESTER_LB06_TH_C04 := 46574,
	TESTER_LB06_TH_D01 := 46581,
	TESTER_LB06_TH_D02 := 46582,
	TESTER_LB06_TH_D03 := 46583,
	TESTER_LB06_TH_D04 := 46584,
	TESTER_LC01 := 47000,
	TESTER_LC01_SOCKET_A01 := 47001,
	TESTER_LC01_SOCKET_A02 := 47002,
	TESTER_LC01_SOCKET_A03 := 47003,
	TESTER_LC01_SOCKET_A04 := 47004,
	TESTER_LC01_SOCKET_B01 := 47011,
	TESTER_LC01_SOCKET_B02 := 47012,
	TESTER_LC01_SOCKET_B03 := 47013,
	TESTER_LC01_SOCKET_B04 := 47014,
	TESTER_LC01_SOCKET_C01 := 47021,
	TESTER_LC01_SOCKET_C02 := 47022,
	TESTER_LC01_SOCKET_C03 := 47023,
	TESTER_LC01_SOCKET_C04 := 47024,
	TESTER_LC01_SOCKET_D01 := 47031,
	TESTER_LC01_SOCKET_D02 := 47032,
	TESTER_LC01_SOCKET_D03 := 47033,
	TESTER_LC01_SOCKET_D04 := 47034,
	TESTER_LC01_TH_A01 := 47051,
	TESTER_LC01_TH_A02 := 47052,
	TESTER_LC01_TH_A03 := 47053,
	TESTER_LC01_TH_A04 := 47054,
	TESTER_LC01_TH_B01 := 47061,
	TESTER_LC01_TH_B02 := 47062,
	TESTER_LC01_TH_B03 := 47063,
	TESTER_LC01_TH_B04 := 47064,
	TESTER_LC01_TH_C01 := 47071,
	TESTER_LC01_TH_C02 := 47072,
	TESTER_LC01_TH_C03 := 47073,
	TESTER_LC01_TH_C04 := 47074,
	TESTER_LC01_TH_D01 := 47081,
	TESTER_LC01_TH_D02 := 47082,
	TESTER_LC01_TH_D03 := 47083,
	TESTER_LC01_TH_D04 := 47084,
	TESTER_LC02 := 47100,
	TESTER_LC02_SOCKET_A01 := 47101,
	TESTER_LC02_SOCKET_A02 := 47102,
	TESTER_LC02_SOCKET_A03 := 47103,
	TESTER_LC02_SOCKET_A04 := 47104,
	TESTER_LC02_SOCKET_B01 := 47111,
	TESTER_LC02_SOCKET_B02 := 47112,
	TESTER_LC02_SOCKET_B03 := 47113,
	TESTER_LC02_SOCKET_B04 := 47114,
	TESTER_LC02_SOCKET_C01 := 47121,
	TESTER_LC02_SOCKET_C02 := 47122,
	TESTER_LC02_SOCKET_C03 := 47123,
	TESTER_LC02_SOCKET_C04 := 47124,
	TESTER_LC02_SOCKET_D01 := 47131,
	TESTER_LC02_SOCKET_D02 := 47132,
	TESTER_LC02_SOCKET_D03 := 47133,
	TESTER_LC02_SOCKET_D04 := 47134,
	TESTER_LC02_TH_A01 := 47151,
	TESTER_LC02_TH_A02 := 47152,
	TESTER_LC02_TH_A03 := 47153,
	TESTER_LC02_TH_A04 := 47154,
	TESTER_LC02_TH_B01 := 47161,
	TESTER_LC02_TH_B02 := 47162,
	TESTER_LC02_TH_B03 := 47163,
	TESTER_LC02_TH_B04 := 47164,
	TESTER_LC02_TH_C01 := 47171,
	TESTER_LC02_TH_C02 := 47172,
	TESTER_LC02_TH_C03 := 47173,
	TESTER_LC02_TH_C04 := 47174,
	TESTER_LC02_TH_D01 := 47181,
	TESTER_LC02_TH_D02 := 47182,
	TESTER_LC02_TH_D03 := 47183,
	TESTER_LC02_TH_D04 := 47184,
	TESTER_LC03 := 47200,
	TESTER_LC03_SOCKET_A01 := 47201,
	TESTER_LC03_SOCKET_A02 := 47202,
	TESTER_LC03_SOCKET_A03 := 47203,
	TESTER_LC03_SOCKET_A04 := 47204,
	TESTER_LC03_SOCKET_B01 := 47211,
	TESTER_LC03_SOCKET_B02 := 47212,
	TESTER_LC03_SOCKET_B03 := 47213,
	TESTER_LC03_SOCKET_B04 := 47214,
	TESTER_LC03_SOCKET_C01 := 47221,
	TESTER_LC03_SOCKET_C02 := 47222,
	TESTER_LC03_SOCKET_C03 := 47223,
	TESTER_LC03_SOCKET_C04 := 47224,
	TESTER_LC03_SOCKET_D01 := 47231,
	TESTER_LC03_SOCKET_D02 := 47232,
	TESTER_LC03_SOCKET_D03 := 47233,
	TESTER_LC03_SOCKET_D04 := 47234,
	TESTER_LC03_TH_A01 := 47251,
	TESTER_LC03_TH_A02 := 47252,
	TESTER_LC03_TH_A03 := 47253,
	TESTER_LC03_TH_A04 := 47254,
	TESTER_LC03_TH_B01 := 47261,
	TESTER_LC03_TH_B02 := 47262,
	TESTER_LC03_TH_B03 := 47263,
	TESTER_LC03_TH_B04 := 47264,
	TESTER_LC03_TH_C01 := 47271,
	TESTER_LC03_TH_C02 := 47272,
	TESTER_LC03_TH_C03 := 47273,
	TESTER_LC03_TH_C04 := 47274,
	TESTER_LC03_TH_D01 := 47281,
	TESTER_LC03_TH_D02 := 47282,
	TESTER_LC03_TH_D03 := 47283,
	TESTER_LC03_TH_D04 := 47284,
	TESTER_LC04 := 47300,
	TESTER_LC04_SOCKET_A01 := 47301,
	TESTER_LC04_SOCKET_A02 := 47302,
	TESTER_LC04_SOCKET_A03 := 47303,
	TESTER_LC04_SOCKET_A04 := 47304,
	TESTER_LC04_SOCKET_B01 := 47311,
	TESTER_LC04_SOCKET_B02 := 47312,
	TESTER_LC04_SOCKET_B03 := 47313,
	TESTER_LC04_SOCKET_B04 := 47314,
	TESTER_LC04_SOCKET_C01 := 47321,
	TESTER_LC04_SOCKET_C02 := 47322,
	TESTER_LC04_SOCKET_C03 := 47323,
	TESTER_LC04_SOCKET_C04 := 47324,
	TESTER_LC04_SOCKET_D01 := 47331,
	TESTER_LC04_SOCKET_D02 := 47332,
	TESTER_LC04_SOCKET_D03 := 47333,
	TESTER_LC04_SOCKET_D04 := 47334,
	TESTER_LC04_TH_A01 := 47351,
	TESTER_LC04_TH_A02 := 47352,
	TESTER_LC04_TH_A03 := 47353,
	TESTER_LC04_TH_A04 := 47354,
	TESTER_LC04_TH_B01 := 47361,
	TESTER_LC04_TH_B02 := 47362,
	TESTER_LC04_TH_B03 := 47363,
	TESTER_LC04_TH_B04 := 47364,
	TESTER_LC04_TH_C01 := 47371,
	TESTER_LC04_TH_C02 := 47372,
	TESTER_LC04_TH_C03 := 47373,
	TESTER_LC04_TH_C04 := 47374,
	TESTER_LC04_TH_D01 := 47381,
	TESTER_LC04_TH_D02 := 47382,
	TESTER_LC04_TH_D03 := 47383,
	TESTER_LC04_TH_D04 := 47384,
	TESTER_LC05 := 47400,
	TESTER_LC05_SOCKET_A01 := 47401,
	TESTER_LC05_SOCKET_A02 := 47402,
	TESTER_LC05_SOCKET_A03 := 47403,
	TESTER_LC05_SOCKET_A04 := 47404,
	TESTER_LC05_SOCKET_B01 := 47411,
	TESTER_LC05_SOCKET_B02 := 47412,
	TESTER_LC05_SOCKET_B03 := 47413,
	TESTER_LC05_SOCKET_B04 := 47414,
	TESTER_LC05_SOCKET_C01 := 47421,
	TESTER_LC05_SOCKET_C02 := 47422,
	TESTER_LC05_SOCKET_C03 := 47423,
	TESTER_LC05_SOCKET_C04 := 47424,
	TESTER_LC05_SOCKET_D01 := 47431,
	TESTER_LC05_SOCKET_D02 := 47432,
	TESTER_LC05_SOCKET_D03 := 47433,
	TESTER_LC05_SOCKET_D04 := 47434,
	TESTER_LC05_TH_A01 := 47451,
	TESTER_LC05_TH_A02 := 47452,
	TESTER_LC05_TH_A03 := 47453,
	TESTER_LC05_TH_A04 := 47454,
	TESTER_LC05_TH_B01 := 47461,
	TESTER_LC05_TH_B02 := 47462,
	TESTER_LC05_TH_B03 := 47463,
	TESTER_LC05_TH_B04 := 47464,
	TESTER_LC05_TH_C01 := 47471,
	TESTER_LC05_TH_C02 := 47472,
	TESTER_LC05_TH_C03 := 47473,
	TESTER_LC05_TH_C04 := 47474,
	TESTER_LC05_TH_D01 := 47481,
	TESTER_LC05_TH_D02 := 47482,
	TESTER_LC05_TH_D03 := 47483,
	TESTER_LC05_TH_D04 := 47484,
	TESTER_LC06 := 47500,
	TESTER_LC06_SOCKET_A01 := 47501,
	TESTER_LC06_SOCKET_A02 := 47502,
	TESTER_LC06_SOCKET_A03 := 47503,
	TESTER_LC06_SOCKET_A04 := 47504,
	TESTER_LC06_SOCKET_B01 := 47511,
	TESTER_LC06_SOCKET_B02 := 47512,
	TESTER_LC06_SOCKET_B03 := 47513,
	TESTER_LC06_SOCKET_B04 := 47514,
	TESTER_LC06_SOCKET_C01 := 47521,
	TESTER_LC06_SOCKET_C02 := 47522,
	TESTER_LC06_SOCKET_C03 := 47523,
	TESTER_LC06_SOCKET_C04 := 47524,
	TESTER_LC06_SOCKET_D01 := 47531,
	TESTER_LC06_SOCKET_D02 := 47532,
	TESTER_LC06_SOCKET_D03 := 47533,
	TESTER_LC06_SOCKET_D04 := 47534,
	TESTER_LC06_TH_A01 := 47551,
	TESTER_LC06_TH_A02 := 47552,
	TESTER_LC06_TH_A03 := 47553,
	TESTER_LC06_TH_A04 := 47554,
	TESTER_LC06_TH_B01 := 47561,
	TESTER_LC06_TH_B02 := 47562,
	TESTER_LC06_TH_B03 := 47563,
	TESTER_LC06_TH_B04 := 47564,
	TESTER_LC06_TH_C01 := 47571,
	TESTER_LC06_TH_C02 := 47572,
	TESTER_LC06_TH_C03 := 47573,
	TESTER_LC06_TH_C04 := 47574,
	TESTER_LC06_TH_D01 := 47581,
	TESTER_LC06_TH_D02 := 47582,
	TESTER_LC06_TH_D03 := 47583,
	TESTER_LC06_TH_D04 := 47584,
	TESTER_RA01 := 50000,
	TESTER_RA01_SOCKET_A01 := 50001,
	TESTER_RA01_SOCKET_A02 := 50002,
	TESTER_RA01_SOCKET_A03 := 50003,
	TESTER_RA01_SOCKET_A04 := 50004,
	TESTER_RA01_SOCKET_B01 := 50011,
	TESTER_RA01_SOCKET_B02 := 50012,
	TESTER_RA01_SOCKET_B03 := 50013,
	TESTER_RA01_SOCKET_B04 := 50014,
	TESTER_RA01_SOCKET_C01 := 50021,
	TESTER_RA01_SOCKET_C02 := 50022,
	TESTER_RA01_SOCKET_C03 := 50023,
	TESTER_RA01_SOCKET_C04 := 50024,
	TESTER_RA01_SOCKET_D01 := 50031,
	TESTER_RA01_SOCKET_D02 := 50032,
	TESTER_RA01_SOCKET_D03 := 50033,
	TESTER_RA01_SOCKET_D04 := 50034,
	TESTER_RA01_TH_A01 := 50051,
	TESTER_RA01_TH_A02 := 50052,
	TESTER_RA01_TH_A03 := 50053,
	TESTER_RA01_TH_A04 := 50054,
	TESTER_RA01_TH_B01 := 50061,
	TESTER_RA01_TH_B02 := 50062,
	TESTER_RA01_TH_B03 := 50063,
	TESTER_RA01_TH_B04 := 50064,
	TESTER_RA01_TH_C01 := 50071,
	TESTER_RA01_TH_C02 := 50072,
	TESTER_RA01_TH_C03 := 50073,
	TESTER_RA01_TH_C04 := 50074,
	TESTER_RA01_TH_D01 := 50081,
	TESTER_RA01_TH_D02 := 50082,
	TESTER_RA01_TH_D03 := 50083,
	TESTER_RA01_TH_D04 := 50084,
	TESTER_RA02 := 50100,
	TESTER_RA02_SOCKET_A01 := 50101,
	TESTER_RA02_SOCKET_A02 := 50102,
	TESTER_RA02_SOCKET_A03 := 50103,
	TESTER_RA02_SOCKET_A04 := 50104,
	TESTER_RA02_SOCKET_B01 := 50111,
	TESTER_RA02_SOCKET_B02 := 50112,
	TESTER_RA02_SOCKET_B03 := 50113,
	TESTER_RA02_SOCKET_B04 := 50114,
	TESTER_RA02_SOCKET_C01 := 50121,
	TESTER_RA02_SOCKET_C02 := 50122,
	TESTER_RA02_SOCKET_C03 := 50123,
	TESTER_RA02_SOCKET_C04 := 50124,
	TESTER_RA02_SOCKET_D01 := 50131,
	TESTER_RA02_SOCKET_D02 := 50132,
	TESTER_RA02_SOCKET_D03 := 50133,
	TESTER_RA02_SOCKET_D04 := 50134,
	TESTER_RA02_TH_A01 := 50151,
	TESTER_RA02_TH_A02 := 50152,
	TESTER_RA02_TH_A03 := 50153,
	TESTER_RA02_TH_A04 := 50154,
	TESTER_RA02_TH_B01 := 50161,
	TESTER_RA02_TH_B02 := 50162,
	TESTER_RA02_TH_B03 := 50163,
	TESTER_RA02_TH_B04 := 50164,
	TESTER_RA02_TH_C01 := 50171,
	TESTER_RA02_TH_C02 := 50172,
	TESTER_RA02_TH_C03 := 50173,
	TESTER_RA02_TH_C04 := 50174,
	TESTER_RA02_TH_D01 := 50181,
	TESTER_RA02_TH_D02 := 50182,
	TESTER_RA02_TH_D03 := 50183,
	TESTER_RA02_TH_D04 := 50184,
	TESTER_RA03 := 50200,
	TESTER_RA03_SOCKET_A01 := 50201,
	TESTER_RA03_SOCKET_A02 := 50202,
	TESTER_RA03_SOCKET_A03 := 50203,
	TESTER_RA03_SOCKET_A04 := 50204,
	TESTER_RA03_SOCKET_B01 := 50211,
	TESTER_RA03_SOCKET_B02 := 50212,
	TESTER_RA03_SOCKET_B03 := 50213,
	TESTER_RA03_SOCKET_B04 := 50214,
	TESTER_RA03_SOCKET_C01 := 50221,
	TESTER_RA03_SOCKET_C02 := 50222,
	TESTER_RA03_SOCKET_C03 := 50223,
	TESTER_RA03_SOCKET_C04 := 50224,
	TESTER_RA03_SOCKET_D01 := 50231,
	TESTER_RA03_SOCKET_D02 := 50232,
	TESTER_RA03_SOCKET_D03 := 50233,
	TESTER_RA03_SOCKET_D04 := 50234,
	TESTER_RA03_TH_A01 := 50251,
	TESTER_RA03_TH_A02 := 50252,
	TESTER_RA03_TH_A03 := 50253,
	TESTER_RA03_TH_A04 := 50254,
	TESTER_RA03_TH_B01 := 50261,
	TESTER_RA03_TH_B02 := 50262,
	TESTER_RA03_TH_B03 := 50263,
	TESTER_RA03_TH_B04 := 50264,
	TESTER_RA03_TH_C01 := 50271,
	TESTER_RA03_TH_C02 := 50272,
	TESTER_RA03_TH_C03 := 50273,
	TESTER_RA03_TH_C04 := 50274,
	TESTER_RA03_TH_D01 := 50281,
	TESTER_RA03_TH_D02 := 50282,
	TESTER_RA03_TH_D03 := 50283,
	TESTER_RA03_TH_D04 := 50284,
	TESTER_RA04 := 50300,
	TESTER_RA04_SOCKET_A01 := 50301,
	TESTER_RA04_SOCKET_A02 := 50302,
	TESTER_RA04_SOCKET_A03 := 50303,
	TESTER_RA04_SOCKET_A04 := 50304,
	TESTER_RA04_SOCKET_B01 := 50311,
	TESTER_RA04_SOCKET_B02 := 50312,
	TESTER_RA04_SOCKET_B03 := 50313,
	TESTER_RA04_SOCKET_B04 := 50314,
	TESTER_RA04_SOCKET_C01 := 50321,
	TESTER_RA04_SOCKET_C02 := 50322,
	TESTER_RA04_SOCKET_C03 := 50323,
	TESTER_RA04_SOCKET_C04 := 50324,
	TESTER_RA04_SOCKET_D01 := 50331,
	TESTER_RA04_SOCKET_D02 := 50332,
	TESTER_RA04_SOCKET_D03 := 50333,
	TESTER_RA04_SOCKET_D04 := 50334,
	TESTER_RA04_TH_A01 := 50351,
	TESTER_RA04_TH_A02 := 50352,
	TESTER_RA04_TH_A03 := 50353,
	TESTER_RA04_TH_A04 := 50354,
	TESTER_RA04_TH_B01 := 50361,
	TESTER_RA04_TH_B02 := 50362,
	TESTER_RA04_TH_B03 := 50363,
	TESTER_RA04_TH_B04 := 50364,
	TESTER_RA04_TH_C01 := 50371,
	TESTER_RA04_TH_C02 := 50372,
	TESTER_RA04_TH_C03 := 50373,
	TESTER_RA04_TH_C04 := 50374,
	TESTER_RA04_TH_D01 := 50381,
	TESTER_RA04_TH_D02 := 50382,
	TESTER_RA04_TH_D03 := 50383,
	TESTER_RA04_TH_D04 := 50384,
	TESTER_RA05 := 50400,
	TESTER_RA05_SOCKET_A01 := 50401,
	TESTER_RA05_SOCKET_A02 := 50402,
	TESTER_RA05_SOCKET_A03 := 50403,
	TESTER_RA05_SOCKET_A04 := 50404,
	TESTER_RA05_SOCKET_B01 := 50411,
	TESTER_RA05_SOCKET_B02 := 50412,
	TESTER_RA05_SOCKET_B03 := 50413,
	TESTER_RA05_SOCKET_B04 := 50414,
	TESTER_RA05_SOCKET_C01 := 50421,
	TESTER_RA05_SOCKET_C02 := 50422,
	TESTER_RA05_SOCKET_C03 := 50423,
	TESTER_RA05_SOCKET_C04 := 50424,
	TESTER_RA05_SOCKET_D01 := 50431,
	TESTER_RA05_SOCKET_D02 := 50432,
	TESTER_RA05_SOCKET_D03 := 50433,
	TESTER_RA05_SOCKET_D04 := 50434,
	TESTER_RA05_TH_A01 := 50451,
	TESTER_RA05_TH_A02 := 50452,
	TESTER_RA05_TH_A03 := 50453,
	TESTER_RA05_TH_A04 := 50454,
	TESTER_RA05_TH_B01 := 50461,
	TESTER_RA05_TH_B02 := 50462,
	TESTER_RA05_TH_B03 := 50463,
	TESTER_RA05_TH_B04 := 50464,
	TESTER_RA05_TH_C01 := 50471,
	TESTER_RA05_TH_C02 := 50472,
	TESTER_RA05_TH_C03 := 50473,
	TESTER_RA05_TH_C04 := 50474,
	TESTER_RA05_TH_D01 := 50481,
	TESTER_RA05_TH_D02 := 50482,
	TESTER_RA05_TH_D03 := 50483,
	TESTER_RA05_TH_D04 := 50484,
	TESTER_RA06 := 50500,
	TESTER_RA06_SOCKET_A01 := 50501,
	TESTER_RA06_SOCKET_A02 := 50502,
	TESTER_RA06_SOCKET_A03 := 50503,
	TESTER_RA06_SOCKET_A04 := 50504,
	TESTER_RA06_SOCKET_B01 := 50511,
	TESTER_RA06_SOCKET_B02 := 50512,
	TESTER_RA06_SOCKET_B03 := 50513,
	TESTER_RA06_SOCKET_B04 := 50514,
	TESTER_RA06_SOCKET_C01 := 50521,
	TESTER_RA06_SOCKET_C02 := 50522,
	TESTER_RA06_SOCKET_C03 := 50523,
	TESTER_RA06_SOCKET_C04 := 50524,
	TESTER_RA06_SOCKET_D01 := 50531,
	TESTER_RA06_SOCKET_D02 := 50532,
	TESTER_RA06_SOCKET_D03 := 50533,
	TESTER_RA06_SOCKET_D04 := 50534,
	TESTER_RA06_TH_A01 := 50551,
	TESTER_RA06_TH_A02 := 50552,
	TESTER_RA06_TH_A03 := 50553,
	TESTER_RA06_TH_A04 := 50554,
	TESTER_RA06_TH_B01 := 50561,
	TESTER_RA06_TH_B02 := 50562,
	TESTER_RA06_TH_B03 := 50563,
	TESTER_RA06_TH_B04 := 50564,
	TESTER_RA06_TH_C01 := 50571,
	TESTER_RA06_TH_C02 := 50572,
	TESTER_RA06_TH_C03 := 50573,
	TESTER_RA06_TH_C04 := 50574,
	TESTER_RA06_TH_D01 := 50581,
	TESTER_RA06_TH_D02 := 50582,
	TESTER_RA06_TH_D03 := 50583,
	TESTER_RA06_TH_D04 := 50584,
	TESTER_RB01 := 51000,
	TESTER_RB01_SOCKET_A01 := 51001,
	TESTER_RB01_SOCKET_A02 := 51002,
	TESTER_RB01_SOCKET_A03 := 51003,
	TESTER_RB01_SOCKET_A04 := 51004,
	TESTER_RB01_SOCKET_B01 := 51011,
	TESTER_RB01_SOCKET_B02 := 51012,
	TESTER_RB01_SOCKET_B03 := 51013,
	TESTER_RB01_SOCKET_B04 := 51014,
	TESTER_RB01_SOCKET_C01 := 51021,
	TESTER_RB01_SOCKET_C02 := 51022,
	TESTER_RB01_SOCKET_C03 := 51023,
	TESTER_RB01_SOCKET_C04 := 51024,
	TESTER_RB01_SOCKET_D01 := 51031,
	TESTER_RB01_SOCKET_D02 := 51032,
	TESTER_RB01_SOCKET_D03 := 51033,
	TESTER_RB01_SOCKET_D04 := 51034,
	TESTER_RB01_TH_A01 := 51051,
	TESTER_RB01_TH_A02 := 51052,
	TESTER_RB01_TH_A03 := 51053,
	TESTER_RB01_TH_A04 := 51054,
	TESTER_RB01_TH_B01 := 51061,
	TESTER_RB01_TH_B02 := 51062,
	TESTER_RB01_TH_B03 := 51063,
	TESTER_RB01_TH_B04 := 51064,
	TESTER_RB01_TH_C01 := 51071,
	TESTER_RB01_TH_C02 := 51072,
	TESTER_RB01_TH_C03 := 51073,
	TESTER_RB01_TH_C04 := 51074,
	TESTER_RB01_TH_D01 := 51081,
	TESTER_RB01_TH_D02 := 51082,
	TESTER_RB01_TH_D03 := 51083,
	TESTER_RB01_TH_D04 := 51084,
	TESTER_RB02 := 51100,
	TESTER_RB02_SOCKET_A01 := 51101,
	TESTER_RB02_SOCKET_A02 := 51102,
	TESTER_RB02_SOCKET_A03 := 51103,
	TESTER_RB02_SOCKET_A04 := 51104,
	TESTER_RB02_SOCKET_B01 := 51111,
	TESTER_RB02_SOCKET_B02 := 51112,
	TESTER_RB02_SOCKET_B03 := 51113,
	TESTER_RB02_SOCKET_B04 := 51114,
	TESTER_RB02_SOCKET_C01 := 51121,
	TESTER_RB02_SOCKET_C02 := 51122,
	TESTER_RB02_SOCKET_C03 := 51123,
	TESTER_RB02_SOCKET_C04 := 51124,
	TESTER_RB02_SOCKET_D01 := 51131,
	TESTER_RB02_SOCKET_D02 := 51132,
	TESTER_RB02_SOCKET_D03 := 51133,
	TESTER_RB02_SOCKET_D04 := 51134,
	TESTER_RB02_TH_A01 := 51151,
	TESTER_RB02_TH_A02 := 51152,
	TESTER_RB02_TH_A03 := 51153,
	TESTER_RB02_TH_A04 := 51154,
	TESTER_RB02_TH_B01 := 51161,
	TESTER_RB02_TH_B02 := 51162,
	TESTER_RB02_TH_B03 := 51163,
	TESTER_RB02_TH_B04 := 51164,
	TESTER_RB02_TH_C01 := 51171,
	TESTER_RB02_TH_C02 := 51172,
	TESTER_RB02_TH_C03 := 51173,
	TESTER_RB02_TH_C04 := 51174,
	TESTER_RB02_TH_D01 := 51181,
	TESTER_RB02_TH_D02 := 51182,
	TESTER_RB02_TH_D03 := 51183,
	TESTER_RB02_TH_D04 := 51184,
	TESTER_RB03 := 51200,
	TESTER_RB03_SOCKET_A01 := 51201,
	TESTER_RB03_SOCKET_A02 := 51202,
	TESTER_RB03_SOCKET_A03 := 51203,
	TESTER_RB03_SOCKET_A04 := 51204,
	TESTER_RB03_SOCKET_B01 := 51211,
	TESTER_RB03_SOCKET_B02 := 51212,
	TESTER_RB03_SOCKET_B03 := 51213,
	TESTER_RB03_SOCKET_B04 := 51214,
	TESTER_RB03_SOCKET_C01 := 51221,
	TESTER_RB03_SOCKET_C02 := 51222,
	TESTER_RB03_SOCKET_C03 := 51223,
	TESTER_RB03_SOCKET_C04 := 51224,
	TESTER_RB03_SOCKET_D01 := 51231,
	TESTER_RB03_SOCKET_D02 := 51232,
	TESTER_RB03_SOCKET_D03 := 51233,
	TESTER_RB03_SOCKET_D04 := 51234,
	TESTER_RB03_TH_A01 := 51251,
	TESTER_RB03_TH_A02 := 51252,
	TESTER_RB03_TH_A03 := 51253,
	TESTER_RB03_TH_A04 := 51254,
	TESTER_RB03_TH_B01 := 51261,
	TESTER_RB03_TH_B02 := 51262,
	TESTER_RB03_TH_B03 := 51263,
	TESTER_RB03_TH_B04 := 51264,
	TESTER_RB03_TH_C01 := 51271,
	TESTER_RB03_TH_C02 := 51272,
	TESTER_RB03_TH_C03 := 51273,
	TESTER_RB03_TH_C04 := 51274,
	TESTER_RB03_TH_D01 := 51281,
	TESTER_RB03_TH_D02 := 51282,
	TESTER_RB03_TH_D03 := 51283,
	TESTER_RB03_TH_D04 := 51284,
	TESTER_RB04 := 51300,
	TESTER_RB04_SOCKET_A01 := 51301,
	TESTER_RB04_SOCKET_A02 := 51302,
	TESTER_RB04_SOCKET_A03 := 51303,
	TESTER_RB04_SOCKET_A04 := 51304,
	TESTER_RB04_SOCKET_B01 := 51311,
	TESTER_RB04_SOCKET_B02 := 51312,
	TESTER_RB04_SOCKET_B03 := 51313,
	TESTER_RB04_SOCKET_B04 := 51314,
	TESTER_RB04_SOCKET_C01 := 51321,
	TESTER_RB04_SOCKET_C02 := 51322,
	TESTER_RB04_SOCKET_C03 := 51323,
	TESTER_RB04_SOCKET_C04 := 51324,
	TESTER_RB04_SOCKET_D01 := 51331,
	TESTER_RB04_SOCKET_D02 := 51332,
	TESTER_RB04_SOCKET_D03 := 51333,
	TESTER_RB04_SOCKET_D04 := 51334,
	TESTER_RB04_TH_A01 := 51351,
	TESTER_RB04_TH_A02 := 51352,
	TESTER_RB04_TH_A03 := 51353,
	TESTER_RB04_TH_A04 := 51354,
	TESTER_RB04_TH_B01 := 51361,
	TESTER_RB04_TH_B02 := 51362,
	TESTER_RB04_TH_B03 := 51363,
	TESTER_RB04_TH_B04 := 51364,
	TESTER_RB04_TH_C01 := 51371,
	TESTER_RB04_TH_C02 := 51372,
	TESTER_RB04_TH_C03 := 51373,
	TESTER_RB04_TH_C04 := 51374,
	TESTER_RB04_TH_D01 := 51381,
	TESTER_RB04_TH_D02 := 51382,
	TESTER_RB04_TH_D03 := 51383,
	TESTER_RB04_TH_D04 := 51384,
	TESTER_RB05 := 51400,
	TESTER_RB05_SOCKET_A01 := 51401,
	TESTER_RB05_SOCKET_A02 := 51402,
	TESTER_RB05_SOCKET_A03 := 51403,
	TESTER_RB05_SOCKET_A04 := 51404,
	TESTER_RB05_SOCKET_B01 := 51411,
	TESTER_RB05_SOCKET_B02 := 51412,
	TESTER_RB05_SOCKET_B03 := 51413,
	TESTER_RB05_SOCKET_B04 := 51414,
	TESTER_RB05_SOCKET_C01 := 51421,
	TESTER_RB05_SOCKET_C02 := 51422,
	TESTER_RB05_SOCKET_C03 := 51423,
	TESTER_RB05_SOCKET_C04 := 51424,
	TESTER_RB05_SOCKET_D01 := 51431,
	TESTER_RB05_SOCKET_D02 := 51432,
	TESTER_RB05_SOCKET_D03 := 51433,
	TESTER_RB05_SOCKET_D04 := 51434,
	TESTER_RB05_TH_A01 := 51451,
	TESTER_RB05_TH_A02 := 51452,
	TESTER_RB05_TH_A03 := 51453,
	TESTER_RB05_TH_A04 := 51454,
	TESTER_RB05_TH_B01 := 51461,
	TESTER_RB05_TH_B02 := 51462,
	TESTER_RB05_TH_B03 := 51463,
	TESTER_RB05_TH_B04 := 51464,
	TESTER_RB05_TH_C01 := 51471,
	TESTER_RB05_TH_C02 := 51472,
	TESTER_RB05_TH_C03 := 51473,
	TESTER_RB05_TH_C04 := 51474,
	TESTER_RB05_TH_D01 := 51481,
	TESTER_RB05_TH_D02 := 51482,
	TESTER_RB05_TH_D03 := 51483,
	TESTER_RB05_TH_D04 := 51484,
	TESTER_RB06 := 51500,
	TESTER_RB06_SOCKET_A01 := 51501,
	TESTER_RB06_SOCKET_A02 := 51502,
	TESTER_RB06_SOCKET_A03 := 51503,
	TESTER_RB06_SOCKET_A04 := 51504,
	TESTER_RB06_SOCKET_B01 := 51511,
	TESTER_RB06_SOCKET_B02 := 51512,
	TESTER_RB06_SOCKET_B03 := 51513,
	TESTER_RB06_SOCKET_B04 := 51514,
	TESTER_RB06_SOCKET_C01 := 51521,
	TESTER_RB06_SOCKET_C02 := 51522,
	TESTER_RB06_SOCKET_C03 := 51523,
	TESTER_RB06_SOCKET_C04 := 51524,
	TESTER_RB06_SOCKET_D01 := 51531,
	TESTER_RB06_SOCKET_D02 := 51532,
	TESTER_RB06_SOCKET_D03 := 51533,
	TESTER_RB06_SOCKET_D04 := 51534,
	TESTER_RB06_TH_A01 := 51551,
	TESTER_RB06_TH_A02 := 51552,
	TESTER_RB06_TH_A03 := 51553,
	TESTER_RB06_TH_A04 := 51554,
	TESTER_RB06_TH_B01 := 51561,
	TESTER_RB06_TH_B02 := 51562,
	TESTER_RB06_TH_B03 := 51563,
	TESTER_RB06_TH_B04 := 51564,
	TESTER_RB06_TH_C01 := 51571,
	TESTER_RB06_TH_C02 := 51572,
	TESTER_RB06_TH_C03 := 51573,
	TESTER_RB06_TH_C04 := 51574,
	TESTER_RB06_TH_D01 := 51581,
	TESTER_RB06_TH_D02 := 51582,
	TESTER_RB06_TH_D03 := 51583,
	TESTER_RB06_TH_D04 := 51584,
	TESTER_RC01 := 52000,
	TESTER_RC01_SOCKET_A01 := 52001,
	TESTER_RC01_SOCKET_A02 := 52002,
	TESTER_RC01_SOCKET_A03 := 52003,
	TESTER_RC01_SOCKET_A04 := 52004,
	TESTER_RC01_SOCKET_B01 := 52011,
	TESTER_RC01_SOCKET_B02 := 52012,
	TESTER_RC01_SOCKET_B03 := 52013,
	TESTER_RC01_SOCKET_B04 := 52014,
	TESTER_RC01_SOCKET_C01 := 52021,
	TESTER_RC01_SOCKET_C02 := 52022,
	TESTER_RC01_SOCKET_C03 := 52023,
	TESTER_RC01_SOCKET_C04 := 52024,
	TESTER_RC01_SOCKET_D01 := 52031,
	TESTER_RC01_SOCKET_D02 := 52032,
	TESTER_RC01_SOCKET_D03 := 52033,
	TESTER_RC01_SOCKET_D04 := 52034,
	TESTER_RC01_TH_A01 := 52051,
	TESTER_RC01_TH_A02 := 52052,
	TESTER_RC01_TH_A03 := 52053,
	TESTER_RC01_TH_A04 := 52054,
	TESTER_RC01_TH_B01 := 52061,
	TESTER_RC01_TH_B02 := 52062,
	TESTER_RC01_TH_B03 := 52063,
	TESTER_RC01_TH_B04 := 52064,
	TESTER_RC01_TH_C01 := 52071,
	TESTER_RC01_TH_C02 := 52072,
	TESTER_RC01_TH_C03 := 52073,
	TESTER_RC01_TH_C04 := 52074,
	TESTER_RC01_TH_D01 := 52081,
	TESTER_RC01_TH_D02 := 52082,
	TESTER_RC01_TH_D03 := 52083,
	TESTER_RC01_TH_D04 := 52084,
	TESTER_RC02 := 52100,
	TESTER_RC02_SOCKET_A01 := 52101,
	TESTER_RC02_SOCKET_A02 := 52102,
	TESTER_RC02_SOCKET_A03 := 52103,
	TESTER_RC02_SOCKET_A04 := 52104,
	TESTER_RC02_SOCKET_B01 := 52111,
	TESTER_RC02_SOCKET_B02 := 52112,
	TESTER_RC02_SOCKET_B03 := 52113,
	TESTER_RC02_SOCKET_B04 := 52114,
	TESTER_RC02_SOCKET_C01 := 52121,
	TESTER_RC02_SOCKET_C02 := 52122,
	TESTER_RC02_SOCKET_C03 := 52123,
	TESTER_RC02_SOCKET_C04 := 52124,
	TESTER_RC02_SOCKET_D01 := 52131,
	TESTER_RC02_SOCKET_D02 := 52132,
	TESTER_RC02_SOCKET_D03 := 52133,
	TESTER_RC02_SOCKET_D04 := 52134,
	TESTER_RC02_TH_A01 := 52151,
	TESTER_RC02_TH_A02 := 52152,
	TESTER_RC02_TH_A03 := 52153,
	TESTER_RC02_TH_A04 := 52154,
	TESTER_RC02_TH_B01 := 52161,
	TESTER_RC02_TH_B02 := 52162,
	TESTER_RC02_TH_B03 := 52163,
	TESTER_RC02_TH_B04 := 52164,
	TESTER_RC02_TH_C01 := 52171,
	TESTER_RC02_TH_C02 := 52172,
	TESTER_RC02_TH_C03 := 52173,
	TESTER_RC02_TH_C04 := 52174,
	TESTER_RC02_TH_D01 := 52181,
	TESTER_RC02_TH_D02 := 52182,
	TESTER_RC02_TH_D03 := 52183,
	TESTER_RC02_TH_D04 := 52184,
	TESTER_RC03 := 52200,
	TESTER_RC03_SOCKET_A01 := 52201,
	TESTER_RC03_SOCKET_A02 := 52202,
	TESTER_RC03_SOCKET_A03 := 52203,
	TESTER_RC03_SOCKET_A04 := 52204,
	TESTER_RC03_SOCKET_B01 := 52211,
	TESTER_RC03_SOCKET_B02 := 52212,
	TESTER_RC03_SOCKET_B03 := 52213,
	TESTER_RC03_SOCKET_B04 := 52214,
	TESTER_RC03_SOCKET_C01 := 52221,
	TESTER_RC03_SOCKET_C02 := 52222,
	TESTER_RC03_SOCKET_C03 := 52223,
	TESTER_RC03_SOCKET_C04 := 52224,
	TESTER_RC03_SOCKET_D01 := 52231,
	TESTER_RC03_SOCKET_D02 := 52232,
	TESTER_RC03_SOCKET_D03 := 52233,
	TESTER_RC03_SOCKET_D04 := 52234,
	TESTER_RC03_TH_A01 := 52251,
	TESTER_RC03_TH_A02 := 52252,
	TESTER_RC03_TH_A03 := 52253,
	TESTER_RC03_TH_A04 := 52254,
	TESTER_RC03_TH_B01 := 52261,
	TESTER_RC03_TH_B02 := 52262,
	TESTER_RC03_TH_B03 := 52263,
	TESTER_RC03_TH_B04 := 52264,
	TESTER_RC03_TH_C01 := 52271,
	TESTER_RC03_TH_C02 := 52272,
	TESTER_RC03_TH_C03 := 52273,
	TESTER_RC03_TH_C04 := 52274,
	TESTER_RC03_TH_D01 := 52281,
	TESTER_RC03_TH_D02 := 52282,
	TESTER_RC03_TH_D03 := 52283,
	TESTER_RC03_TH_D04 := 52284,
	TESTER_RC04 := 52300,
	TESTER_RC04_SOCKET_A01 := 52301,
	TESTER_RC04_SOCKET_A02 := 52302,
	TESTER_RC04_SOCKET_A03 := 52303,
	TESTER_RC04_SOCKET_A04 := 52304,
	TESTER_RC04_SOCKET_B01 := 52311,
	TESTER_RC04_SOCKET_B02 := 52312,
	TESTER_RC04_SOCKET_B03 := 52313,
	TESTER_RC04_SOCKET_B04 := 52314,
	TESTER_RC04_SOCKET_C01 := 52321,
	TESTER_RC04_SOCKET_C02 := 52322,
	TESTER_RC04_SOCKET_C03 := 52323,
	TESTER_RC04_SOCKET_C04 := 52324,
	TESTER_RC04_SOCKET_D01 := 52331,
	TESTER_RC04_SOCKET_D02 := 52332,
	TESTER_RC04_SOCKET_D03 := 52333,
	TESTER_RC04_SOCKET_D04 := 52334,
	TESTER_RC04_TH_A01 := 52351,
	TESTER_RC04_TH_A02 := 52352,
	TESTER_RC04_TH_A03 := 52353,
	TESTER_RC04_TH_A04 := 52354,
	TESTER_RC04_TH_B01 := 52361,
	TESTER_RC04_TH_B02 := 52362,
	TESTER_RC04_TH_B03 := 52363,
	TESTER_RC04_TH_B04 := 52364,
	TESTER_RC04_TH_C01 := 52371,
	TESTER_RC04_TH_C02 := 52372,
	TESTER_RC04_TH_C03 := 52373,
	TESTER_RC04_TH_C04 := 52374,
	TESTER_RC04_TH_D01 := 52381,
	TESTER_RC04_TH_D02 := 52382,
	TESTER_RC04_TH_D03 := 52383,
	TESTER_RC04_TH_D04 := 52384,
	TESTER_RC05 := 52400,
	TESTER_RC05_SOCKET_A01 := 52401,
	TESTER_RC05_SOCKET_A02 := 52402,
	TESTER_RC05_SOCKET_A03 := 52403,
	TESTER_RC05_SOCKET_A04 := 52404,
	TESTER_RC05_SOCKET_B01 := 52411,
	TESTER_RC05_SOCKET_B02 := 52412,
	TESTER_RC05_SOCKET_B03 := 52413,
	TESTER_RC05_SOCKET_B04 := 52414,
	TESTER_RC05_SOCKET_C01 := 52421,
	TESTER_RC05_SOCKET_C02 := 52422,
	TESTER_RC05_SOCKET_C03 := 52423,
	TESTER_RC05_SOCKET_C04 := 52424,
	TESTER_RC05_SOCKET_D01 := 52431,
	TESTER_RC05_SOCKET_D02 := 52432,
	TESTER_RC05_SOCKET_D03 := 52433,
	TESTER_RC05_SOCKET_D04 := 52434,
	TESTER_RC05_TH_A01 := 52451,
	TESTER_RC05_TH_A02 := 52452,
	TESTER_RC05_TH_A03 := 52453,
	TESTER_RC05_TH_A04 := 52454,
	TESTER_RC05_TH_B01 := 52461,
	TESTER_RC05_TH_B02 := 52462,
	TESTER_RC05_TH_B03 := 52463,
	TESTER_RC05_TH_B04 := 52464,
	TESTER_RC05_TH_C01 := 52471,
	TESTER_RC05_TH_C02 := 52472,
	TESTER_RC05_TH_C03 := 52473,
	TESTER_RC05_TH_C04 := 52474,
	TESTER_RC05_TH_D01 := 52481,
	TESTER_RC05_TH_D02 := 52482,
	TESTER_RC05_TH_D03 := 52483,
	TESTER_RC05_TH_D04 := 52484,
	TESTER_RC06 := 52500,
	TESTER_RC06_SOCKET_A01 := 52501,
	TESTER_RC06_SOCKET_A02 := 52502,
	TESTER_RC06_SOCKET_A03 := 52503,
	TESTER_RC06_SOCKET_A04 := 52504,
	TESTER_RC06_SOCKET_B01 := 52511,
	TESTER_RC06_SOCKET_B02 := 52512,
	TESTER_RC06_SOCKET_B03 := 52513,
	TESTER_RC06_SOCKET_B04 := 52514,
	TESTER_RC06_SOCKET_C01 := 52521,
	TESTER_RC06_SOCKET_C02 := 52522,
	TESTER_RC06_SOCKET_C03 := 52523,
	TESTER_RC06_SOCKET_C04 := 52524,
	TESTER_RC06_SOCKET_D01 := 52531,
	TESTER_RC06_SOCKET_D02 := 52532,
	TESTER_RC06_SOCKET_D03 := 52533,
	TESTER_RC06_SOCKET_D04 := 52534,
	TESTER_RC06_TH_A01 := 52551,
	TESTER_RC06_TH_A02 := 52552,
	TESTER_RC06_TH_A03 := 52553,
	TESTER_RC06_TH_A04 := 52554,
	TESTER_RC06_TH_B01 := 52561,
	TESTER_RC06_TH_B02 := 52562,
	TESTER_RC06_TH_B03 := 52563,
	TESTER_RC06_TH_B04 := 52564,
	TESTER_RC06_TH_C01 := 52571,
	TESTER_RC06_TH_C02 := 52572,
	TESTER_RC06_TH_C03 := 52573,
	TESTER_RC06_TH_C04 := 52574,
	TESTER_RC06_TH_D01 := 52581,
	TESTER_RC06_TH_D02 := 52582,
	TESTER_RC06_TH_D03 := 52583,
	TESTER_RC06_TH_D04 := 52584
*)
)dint;
END_TYPE

(* stored: Version 1.1.0.1, ProductVersion 3.1.4022.12
   DUT E_ModuleID: Id {e736d1ab-da9a-4f9c-8978-6a05e844ef5a} *)
